   1:  PR[91,2] = PR[90,2] + -5.952;
   1:  PR[91,3] = PR[90,3] + 71.100;
   1:L PR[91] R[100]mm/sec CNT100;
   1:  PR[91,1] = PR[90,1] + 75.021;
   1:  PR[91,2] = PR[90,2] + -5.106;
   1:  PR[91,3] = PR[90,3] + 71.120;
   1:L PR[91] R[100]mm/sec CNT100;
   1:  PR[91,1] = PR[90,1] + 75.710;
   1:  PR[91,2] = PR[90,2] + -0.815;
   1:  PR[91,3] = PR[90,3] + 71.123;
   1:L PR[91] R[100]mm/sec CNT100;
   1:  PR[91,1] = PR[90,1] + 75.480;
   1:  PR[91,2] = PR[90,2] + 0.111;
   1:  PR[91,3] = PR[90,3] + 71.139;
   1:L PR[91] R[100]mm/sec CNT100;
   1:  PR[91,1] = PR[90,1] + 74.909;
   1:  PR[91,2] = PR[90,2] + 4.493;
   1:  PR[91,3] = PR[90,3] + 71.143;
   1:L PR[91] R[100]mm/sec CNT100;
   1:  PR[91,1] = PR[90,1] + 72.862;
   1:  PR[91,2] = PR[90,2] + 9.573;
   1:  PR[91,3] = PR[90,3] + 71.159;
   1:L PR[91] R[100]mm/sec CNT100;
   1:  PR[91,1] = PR[90,1] + 71.941;
   1:  PR[91,2] = PR[90,2] + 10.859;
   1:  PR[91,3] = PR[90,3] + 71.179;
   1:L PR[91] R[100]mm/sec CNT100;
   1:  PR[91,1] = PR[90,1] + 69.608;
   1:  PR[91,2] = PR[90,2] + 13.845;
   1:  PR[91,3] = PR[90,3] + 71.185;
   1:L PR[91] R[100]mm/sec CNT100;
   1:  PR[91,1] = PR[90,1] + 69.298;
   1:  PR[91,2] = PR[90,2] + 14.226;
   1:  PR[91,3] = PR[90,3] + 71.199;
   1:L PR[91] R[100]mm/sec CNT100;
   1:  PR[91,1] = PR[90,1] + 68.582;
   1:  PR[91,2] = PR[90,2] + 14.856;
   1:  PR[91,3] = PR[90,3] + 71.201;
   1:L PR[91] R[100]mm/sec CNT100;
   1:  PR[91,1] = PR[90,1] + 64.894;
   1:  PR[91,2] = PR[90,2] + 17.899;
   1:  PR[91,3] = PR[90,3] + 71.204;
   1:L PR[91] R[100]mm/sec CNT100;
   1:  PR[91,1] = PR[90,1] + 62.420;
   1:  PR[91,2] = PR[90,2] + 19.477;
   1:  PR[91,3] = PR[90,3] + 71.222;
   1:L PR[91] R[100]mm/sec CNT100;
   1:  PR[91,1] = PR[90,1] + 60.608;
   1:  PR[91,2] = PR[90,2] + 20.459;
   1:  PR[91,3] = PR[90,3] + 71.233;
   1:L PR[91] R[100]mm/sec CNT100;
   1:  PR[91,1] = PR[90,1] + 56.591;
   1:  PR[91,2] = PR[90,2] + 22.307;
   1:  PR[91,3] = PR[90,3] + 71.240;
   1:L PR[91] R[100]mm/sec CNT100;
   1:  PR[91,1] = PR[90,1] + 54.711;
   1:  PR[91,2] = PR[90,2] + 22.922;
   1:  PR[91,3] = PR[90,3] + 71.256;
   1:L PR[91] R[100]mm/sec CNT100;
   1:  PR[91,1] = PR[90,1] + 52.146;
   1:  PR[91,2] = PR[90,2] + 23.718;
   1:  PR[91,3] = PR[90,3] + 71.264;
   1:L PR[91] R[100]mm/sec CNT100;
   1:  PR[91,1] = PR[90,1] + 51.088;
   1:  PR[91,2] = PR[90,2] + 23.935;
   1:  PR[91,3] = PR[90,3] + 71.274;
   1:L PR[91] R[100]mm/sec CNT100;
   1:  PR[91,1] = PR[90,1] + 47.420;
   1:  PR[91,2] = PR[90,2] + 24.845;
   1:  PR[91,3] = PR[90,3] + 71.278;
   1:L PR[91] R[100]mm/sec CNT100;
   1:  PR[91,1] = PR[90,1] + 42.741;
   1:  PR[91,2] = PR[90,2] + 25.473;
   1:  PR[91,3] = PR[90,3] + 71.291;
   1:L PR[91] R[100]mm/sec CNT100;
   1:  PR[91,1] = PR[90,1] + 41.965;
   1:  PR[91,2] = PR[90,2] + 25.566;
   1:  PR[91,3] = PR[90,3] + 71.309;
   1:L PR[91] R[100]mm/sec CNT100;
   1:  PR[91,1] = PR[90,1] + 41.084;
   1:  PR[91,2] = PR[90,2] + 25.570;
   1:  PR[91,3] = PR[90,3] + 71.312;
   1:L PR[91] R[100]mm/sec CNT100;
   1:  PR[91,1] = PR[90,1] + 37.170;
   1:  PR[91,2] = PR[90,2] + 25.636;
   1:  PR[91,3] = PR[90,3] + 71.315;
   1:L PR[91] R[100]mm/sec CNT100;
   1:  PR[91,1] = PR[90,1] + 34.823;
   1:  PR[91,2] = PR[90,2] + 25.445;
   1:  PR[91,3] = PR[90,3] + 71.329;
   1:L PR[91] R[100]mm/sec CNT100;
   1:  PR[91,1] = PR[90,1] + 32.347;
   1:  PR[91,2] = PR[90,2] + 25.103;
   1:  PR[91,3] = PR[90,3] + 71.338;
   1:L PR[91] R[100]mm/sec CNT100;
   1:  PR[91,1] = PR[90,1] + 27.084;
   1:  PR[91,2] = PR[90,2] + 23.838;
   1:  PR[91,3] = PR[90,3] + 71.347;
   1:L PR[91] R[100]mm/sec CNT100;
   1:  PR[91,1] = PR[90,1] + 22.919;
   1:  PR[91,2] = PR[90,2] + 24.474;
   1:  PR[91,3] = PR[90,3] + 71.367;
   1:L PR[91] R[100]mm/sec CNT100;
   1:  PR[91,1] = PR[90,1] + 20.600;
   1:  PR[91,2] = PR[90,2] + 24.549;
   1:  PR[91,3] = PR[90,3] + 71.382;
   1:L PR[91] R[100]mm/sec CNT100;
   1:  PR[91,1] = PR[90,1] + 17.020;
   1:  PR[91,2] = PR[90,2] + 24.403;
   1:  PR[91,3] = PR[90,3] + 71.391;
   1:L PR[91] R[100]mm/sec CNT100;
   1:  PR[91,1] = PR[90,1] + 14.351;
   1:  PR[91,2] = PR[90,2] + 23.828;
   1:  PR[91,3] = PR[90,3] + 71.404;
   1:L PR[91] R[100]mm/sec CNT100;
   1:  PR[91,1] = PR[90,1] + 11.204;
   1:  PR[91,2] = PR[90,2] + 22.970;
   1:  PR[91,3] = PR[90,3] + 71.414;
   1:L PR[91] R[100]mm/sec CNT100;
   1:  PR[91,1] = PR[90,1] + 7.848;
   1:  PR[91,2] = PR[90,2] + 21.430;
   1:  PR[91,3] = PR[90,3] + 71.426;
   1:L PR[91] R[100]mm/sec CNT100;
   1:  PR[91,1] = PR[90,1] + 3.303;
   1:  PR[91,2] = PR[90,2] + 22.600;
   1:  PR[91,3] = PR[90,3] + 71.440;
   1:L PR[91] R[100]mm/sec CNT100;
   1:  PR[91,1] = PR[90,1] + 1.714;
   1:  PR[91,2] = PR[90,2] + 23.052;
   1:  PR[91,3] = PR[90,3] + 71.457;
   1:L PR[91] R[100]mm/sec CNT100;
   1:  PR[91,1] = PR[90,1] + -4.595;
   1:  PR[91,2] = PR[90,2] + 23.619;
   1:  PR[91,3] = PR[90,3] + 71.463;
   1:L PR[91] R[100]mm/sec CNT100;
   1:  PR[91,1] = PR[90,1] + -7.696;
   1:  PR[91,2] = PR[90,2] + 23.369;
   1:  PR[91,3] = PR[90,3] + 71.486;
   1:L PR[91] R[100]mm/sec CNT100;
   1:  PR[91,1] = PR[90,1] + -10.709;
   1:  PR[91,2] = PR[90,2] + 23.080;
   1:  PR[91,3] = PR[90,3] + 71.498;
   1:L PR[91] R[100]mm/sec CNT100;
   1:  PR[91,1] = PR[90,1] + -13.600;
   1:  PR[91,2] = PR[90,2] + 22.402;
   1:  PR[91,3] = PR[90,3] + 71.509;
   1:L PR[91] R[100]mm/sec CNT100;
   1:  PR[91,1] = PR[90,1] + -15.931;
   1:  PR[91,2] = PR[90,2] + 21.755;
   1:  PR[91,3] = PR[90,3] + 71.520;
   1:L PR[91] R[100]mm/sec CNT100;
   1:  PR[91,1] = PR[90,1] + -17.870;
   1:  PR[91,2] = PR[90,2] + 22.083;
   1:  PR[91,3] = PR[90,3] + 71.529;
   1:L PR[91] R[100]mm/sec CNT100;
   1:  PR[91,1] = PR[90,1] + -19.775;
   1:  PR[91,2] = PR[90,2] + 22.343;
   1:  PR[91,3] = PR[90,3] + 71.536;
   1:L PR[91] R[100]mm/sec CNT100;
   1:  PR[91,1] = PR[90,1] + -26.709;
   1:  PR[91,2] = PR[90,2] + 23.102;
   1:  PR[91,3] = PR[90,3] + 71.543;
   1:L PR[91] R[100]mm/sec CNT100;
   1:  PR[91,1] = PR[90,1] + -27.634;
   1:  PR[91,2] = PR[90,2] + 23.219;
   1:  PR[91,3] = PR[90,3] + 71.569;
   1:L PR[91] R[100]mm/sec CNT100;
   1:  PR[91,1] = PR[90,1] + -35.837;
   1:  PR[91,2] = PR[90,2] + 23.471;
   1:  PR[91,3] = PR[90,3] + 71.572;
   1:L PR[91] R[100]mm/sec CNT100;
   1:  PR[91,1] = PR[90,1] + -37.663;
   1:  PR[91,2] = PR[90,2] + 23.575;
   1:  PR[91,3] = PR[90,3] + 71.602;
   1:L PR[91] R[100]mm/sec CNT100;
   1:  PR[91,1] = PR[90,1] + -41.865;
   1:  PR[91,2] = PR[90,2] + 23.392;
   1:  PR[91,3] = PR[90,3] + 71.609;
   1:L PR[91] R[100]mm/sec CNT100;
   1:  PR[91,1] = PR[90,1] + -44.716;
   1:  PR[91,2] = PR[90,2] + 23.204;
   1:  PR[91,3] = PR[90,3] + 71.624;
   1:L PR[91] R[100]mm/sec CNT100;
   1:  PR[91,1] = PR[90,1] + -50.383;
   1:  PR[91,2] = PR[90,2] + 22.257;
   1:  PR[91,3] = PR[90,3] + 71.635;
   1:L PR[91] R[100]mm/sec CNT100;
   1:  PR[91,1] = PR[90,1] + -53.393;
   1:  PR[91,2] = PR[90,2] + 21.640;
   1:  PR[91,3] = PR[90,3] + 71.656;
   1:L PR[91] R[100]mm/sec CNT100;
   1:  PR[91,1] = PR[90,1] + -55.296;
   1:  PR[91,2] = PR[90,2] + 21.017;
   1:  PR[91,3] = PR[90,3] + 71.667;
   1:L PR[91] R[100]mm/sec CNT100;
   1:  PR[91,1] = PR[90,1] + -58.574;
   1:  PR[91,2] = PR[90,2] + 19.824;
   1:  PR[91,3] = PR[90,3] + 71.675;
   1:L PR[91] R[100]mm/sec CNT100;
   1:  PR[91,1] = PR[90,1] + -60.495;
   1:  PR[91,2] = PR[90,2] + 19.070;
   1:  PR[91,3] = PR[90,3] + 71.687;
   1:L PR[91] R[100]mm/sec CNT100;
   1:  PR[91] = PR[90];
   1:  PR[91,1] = PR[90,1] + -64.658;
   1:  PR[91,2] = PR[90,2] + 16.036;
   1:  PR[91,3] = PR[90,3] + 72.995;
   1:L PR[91] R[100]mm/sec CNT100;
   1:  PR[91,1] = PR[90,1] + -66.807;
   1:  PR[91,2] = PR[90,2] + 14.084;
   1:  PR[91,3] = PR[90,3] + 71.717;
   1:L PR[91] R[100]mm/sec CNT100;
   1:  PR[91,1] = PR[90,1] + -68.784;
   1:  PR[91,2] = PR[90,2] + 12.271;
   1:  PR[91,3] = PR[90,3] + 71.728;
   1:L PR[91] R[100]mm/sec CNT100;
   1:  PR[91,1] = PR[90,1] + -71.738;
   1:  PR[91,2] = PR[90,2] + 8.120;
   1:  PR[91,3] = PR[90,3] + 71.738;
   1:L PR[91] R[100]mm/sec CNT100;
   1:  PR[91,1] = PR[90,1] + -73.499;
   1:  PR[91,2] = PR[90,2] + 3.745;
   1:  PR[91,3] = PR[90,3] + 71.757;
   1:L PR[91] R[100]mm/sec CNT100;
   1:  PR[91,1] = PR[90,1] + -74.080;
   1:  PR[91,2] = PR[90,2] + -0.689;
   1:  PR[91,3] = PR[90,3] + 71.774;
   1:L PR[91] R[100]mm/sec CNT100;
   1:  PR[91,1] = PR[90,1] + -73.575;
   1:  PR[91,2] = PR[90,2] + -3.117;
   1:  PR[91,3] = PR[90,3] + 71.791;
   1:L PR[91] R[100]mm/sec CNT100;
   1:  PR[91,1] = PR[90,1] + -73.284;
   1:  PR[91,2] = PR[90,2] + -5.386;
   1:  PR[91,3] = PR[90,3] + 71.800;
   1:L PR[91] R[100]mm/sec CNT100;
   1:  PR[91,1] = PR[90,1] + -72.278;
   1:  PR[91,2] = PR[90,2] + -7.892;
   1:  PR[91,3] = PR[90,3] + 71.808;
   1:L PR[91] R[100]mm/sec CNT100;
   1:  PR[91,1] = PR[90,1] + -71.464;
   1:  PR[91,2] = PR[90,2] + -9.892;
   1:  PR[91,3] = PR[90,3] + 71.818;
   1:L PR[91] R[100]mm/sec CNT100;
   1:  PR[91,1] = PR[90,1] + -68.451;
   1:  PR[91,2] = PR[90,2] + -14.108;
   1:  PR[91,3] = PR[90,3] + 71.826;
   1:L PR[91] R[100]mm/sec CNT100;
   1:  PR[91,1] = PR[90,1] + -64.359;
   1:  PR[91,2] = PR[90,2] + -17.817;
   1:  PR[91,3] = PR[90,3] + 71.846;
   1:L PR[91] R[100]mm/sec CNT100;
   1:  PR[91,1] = PR[90,1] + -59.208;
   1:  PR[91,2] = PR[90,2] + -20.687;
   1:  PR[91,3] = PR[90,3] + 71.866;
   1:L PR[91] R[100]mm/sec CNT100;
   1:  PR[91,1] = PR[90,1] + -56.302;
   1:  PR[91,2] = PR[90,2] + -21.871;
   1:  PR[91,3] = PR[90,3] + 71.888;
   1:L PR[91] R[100]mm/sec CNT100;
   1:  PR[91,1] = PR[90,1] + -53.674;
   1:  PR[91,2] = PR[90,2] + -22.806;
   1:  PR[91,3] = PR[90,3] + 71.900;
   1:L PR[91] R[100]mm/sec CNT100;
   1:  PR[91,1] = PR[90,1] + -49.742;
   1:  PR[91,2] = PR[90,2] + -23.757;
   1:  PR[91,3] = PR[90,3] + 71.910;
   1:L PR[91] R[100]mm/sec CNT100;
   1:  PR[91,1] = PR[90,1] + -47.986;
   1:  PR[91,2] = PR[90,2] + -24.162;
   1:  PR[91,3] = PR[90,3] + 71.925;
   1:L PR[91] R[100]mm/sec CNT100;
   1:  PR[91,1] = PR[90,1] + -46.736;
   1:  PR[91,2] = PR[90,2] + -24.408;
   1:  PR[91,3] = PR[90,3] + 71.932;
   1:L PR[91] R[100]mm/sec CNT100;
   1:  PR[91,1] = PR[90,1] + -42.499;
   1:  PR[91,2] = PR[90,2] + -24.853;
   1:  PR[91,3] = PR[90,3] + 71.937;
   1:L PR[91] R[100]mm/sec CNT100;
   1:  PR[91,1] = PR[90,1] + -37.572;
   1:  PR[91,2] = PR[90,2] + -25.182;
   1:  PR[91,3] = PR[90,3] + 71.952;
   1:L PR[91] R[100]mm/sec CNT100;
   1:  PR[91,1] = PR[90,1] + -36.488;
   1:  PR[91,2] = PR[90,2] + -25.268;
   1:  PR[91,3] = PR[90,3] + 71.971;
   1:L PR[91] R[100]mm/sec CNT100;
   1:  PR[91,1] = PR[90,1] + -35.528;
   1:  PR[91,2] = PR[90,2] + -25.297;
   1:  PR[91,3] = PR[90,3] + 71.975;
   1:L PR[91] R[100]mm/sec CNT100;
   1:  PR[91,1] = PR[90,1] + -30.632;
   1:  PR[91,2] = PR[90,2] + -25.146;
   1:  PR[91,3] = PR[90,3] + 71.978;
   1:L PR[91] R[100]mm/sec CNT100;
   1:  PR[91,1] = PR[90,1] + -24.961;
   1:  PR[91,2] = PR[90,2] + -24.930;
   1:  PR[91,3] = PR[90,3] + 71.996;
   1:L PR[91] R[100]mm/sec CNT100;
   1:  PR[91,1] = PR[90,1] + -17.966;
   1:  PR[91,2] = PR[90,2] + -24.135;
   1:  PR[91,3] = PR[90,3] + 72.017;
   1:L PR[91] R[100]mm/sec CNT100;
   1:  PR[91,1] = PR[90,1] + -17.484;
   1:  PR[91,2] = PR[90,2] + -24.120;
   1:  PR[91,3] = PR[90,3] + 72.044;
   1:L PR[91] R[100]mm/sec CNT100;
   1:  PR[91,1] = PR[90,1] + -14.422;
   1:  PR[91,2] = PR[90,2] + -23.701;
   1:  PR[91,3] = PR[90,3] + 72.045;
   1:L PR[91] R[100]mm/sec CNT100;
   1:  PR[91,1] = PR[90,1] + -10.015;
   1:  PR[91,2] = PR[90,2] + -24.736;
   1:  PR[91,3] = PR[90,3] + 72.057;
   1:L PR[91] R[100]mm/sec CNT100;
   1:  PR[91,1] = PR[90,1] + -5.899;
   1:  PR[91,2] = PR[90,2] + -25.133;
   1:  PR[91,3] = PR[90,3] + 72.074;
   1:L PR[91] R[100]mm/sec CNT100;
   1:  PR[91,1] = PR[90,1] + -3.854;
   1:  PR[91,2] = PR[90,2] + -25.298;
   1:  PR[91,3] = PR[90,3] + 72.089;
   1:L PR[91] R[100]mm/sec CNT100;
   1:  PR[91,1] = PR[90,1] + 2.663;
   1:  PR[91,2] = PR[90,2] + -24.737;
   1:  PR[91,3] = PR[90,3] + 72.097;
   1:L PR[91] R[100]mm/sec CNT100;
   1:  PR[91,1] = PR[90,1] + 8.196;
   1:  PR[91,2] = PR[90,2] + -23.321;
   1:  PR[91,3] = PR[90,3] + 72.121;
   1:L PR[91] R[100]mm/sec CNT100;
   1:  PR[91,1] = PR[90,1] + 11.071;
   1:  PR[91,2] = PR[90,2] + -24.641;
   1:  PR[91,3] = PR[90,3] + 72.142;
   1:L PR[91] R[100]mm/sec CNT100;
   1:  PR[91,1] = PR[90,1] + 13.655;
   1:  PR[91,2] = PR[90,2] + -25.345;
   1:  PR[91,3] = PR[90,3] + 72.154;
   1:L PR[91] R[100]mm/sec CNT100;
   1:  PR[91,1] = PR[90,1] + 16.983;
   1:  PR[91,2] = PR[90,2] + -26.063;
   1:  PR[91,3] = PR[90,3] + 72.164;
   1:L PR[91] R[100]mm/sec CNT100;
   1:  PR[91,1] = PR[90,1] + 19.995;
   1:  PR[91,2] = PR[90,2] + -26.185;
   1:  PR[91,3] = PR[90,3] + 72.176;
   1:L PR[91] R[100]mm/sec CNT100;
   1:  PR[91,1] = PR[90,1] + 22.970;
   1:  PR[91,2] = PR[90,2] + -26.089;
   1:  PR[91,3] = PR[90,3] + 72.188;
   1:L PR[91] R[100]mm/sec CNT100;
   1:  PR[91,1] = PR[90,1] + 26.634;
   1:  PR[91,2] = PR[90,2] + -25.533;
   1:  PR[91,3] = PR[90,3] + 72.199;
   1:L PR[91] R[100]mm/sec CNT100;
   1:  PR[91,1] = PR[90,1] + 29.088;
   1:  PR[91,2] = PR[90,2] + -26.173;
   1:  PR[91,3] = PR[90,3] + 72.212;
   1:L PR[91] R[100]mm/sec CNT100;
   1:  PR[91,1] = PR[90,1] + 31.868;
   1:  PR[91,2] = PR[90,2] + -26.840;
   1:  PR[91,3] = PR[90,3] + 72.222;
   1:L PR[91] R[100]mm/sec CNT100;
   1:  PR[91,1] = PR[90,1] + 33.215;
   1:  PR[91,2] = PR[90,2] + -27.027;
   1:  PR[91,3] = PR[90,3] + 72.232;
   1:L PR[91] R[100]mm/sec CNT100;
   1:  PR[91,1] = PR[90,1] + 36.811;
   1:  PR[91,2] = PR[90,2] + -27.319;
   1:  PR[91,3] = PR[90,3] + 72.237;
   1:L PR[91] R[100]mm/sec CNT100;
   1:  PR[91,1] = PR[90,1] + 40.668;
   1:  PR[91,2] = PR[90,2] + -27.254;
   1:  PR[91,3] = PR[90,3] + 72.251;
   1:L PR[91] R[100]mm/sec CNT100;
   1:  PR[91,1] = PR[90,1] + 41.328;
   1:  PR[91,2] = PR[90,2] + -27.203;
   1:  PR[91,3] = PR[90,3] + 72.265;
   1:L PR[91] R[100]mm/sec CNT100;
   1:  PR[91,1] = PR[90,1] + 42.439;
   1:  PR[91,2] = PR[90,2] + -27.011;
   1:  PR[91,3] = PR[90,3] + 72.268;
   1:L PR[91] R[100]mm/sec CNT100;
   1:  PR[91,1] = PR[90,1] + 46.630;
   1:  PR[91,2] = PR[90,2] + -26.449;
   1:  PR[91,3] = PR[90,3] + 72.272;
   1:L PR[91] R[100]mm/sec CNT100;
   1:  PR[91,1] = PR[90,1] + 50.455;
   1:  PR[91,2] = PR[90,2] + -25.500;
   1:  PR[91,3] = PR[90,3] + 72.288;
   1:L PR[91] R[100]mm/sec CNT100;
   1:  PR[91,1] = PR[90,1] + 51.336;
   1:  PR[91,2] = PR[90,2] + -25.262;
   1:  PR[91,3] = PR[90,3] + 72.302;
   1:L PR[91] R[100]mm/sec CNT100;
   1:  PR[91,1] = PR[90,1] + 52.051;
   1:  PR[91,2] = PR[90,2] + -24.984;
   1:  PR[91,3] = PR[90,3] + 72.306;
   1:L PR[91] R[100]mm/sec CNT100;
   1:  PR[91,1] = PR[90,1] + 55.819;
   1:  PR[91,2] = PR[90,2] + -23.752;
   1:  PR[91,3] = PR[90,3] + 72.308;
   1:L PR[91] R[100]mm/sec CNT100;
   1:  PR[91,1] = PR[90,1] + 60.017;
   1:  PR[91,2] = PR[90,2] + -21.841;
   1:  PR[91,3] = PR[90,3] + 72.323;
   1:L PR[91] R[100]mm/sec CNT100;
   1:  PR[91,1] = PR[90,1] + 60.781;
   1:  PR[91,2] = PR[90,2] + -21.428;
   1:  PR[91,3] = PR[90,3] + 72.340;
   1:L PR[91] R[100]mm/sec CNT100;
   1:  PR[91,1] = PR[90,1] + 64.071;
   1:  PR[91,2] = PR[90,2] + -19.328;
   1:  PR[91,3] = PR[90,3] + 72.343;
   1:L PR[91] R[100]mm/sec CNT100;
   1:  PR[91,1] = PR[90,1] + 66.786;
   1:  PR[91,2] = PR[90,2] + -17.090;
   1:  PR[91,3] = PR[90,3] + 72.358;
   1:L PR[91] R[100]mm/sec CNT100;
   1:  PR[91,1] = PR[90,1] + 68.269;
   1:  PR[91,2] = PR[90,2] + -15.785;
   1:  PR[91,3] = PR[90,3] + 72.371;
   1:L PR[91] R[100]mm/sec CNT100;
   1:  PR[91,1] = PR[90,1] + 71.977;
   1:  PR[91,2] = PR[90,2] + -11.080;
   1:  PR[91,3] = PR[90,3] + 72.378;
   1:L PR[91] R[100]mm/sec CNT100;
   1:  PR[91,1] = PR[90,1] + 72.022;
   1:  PR[91,2] = PR[90,2] + -10.999;
   1:  PR[91,3] = PR[90,3] + 72.401;
   1:L PR[91] R[100]mm/sec CNT100;
   1:  PR[91,1] = PR[90,1] + 73.204;
   1:  PR[91,2] = PR[90,2] + -8.301;
   1:L PR[91] R[100]mm/sec CNT100;
   1:  PR[91,1] = PR[90,1] + 74.139;
   1:  PR[91,2] = PR[90,2] + -5.981;
   1:  PR[91,3] = PR[90,3] + 72.412;
   1:L PR[91] R[100]mm/sec CNT100;
   1:  PR[91,1] = PR[90,1] + 74.388;
   1:  PR[91,2] = PR[90,2] + -4.382;
   1:  PR[91,3] = PR[90,3] + 72.421;
   1:L PR[91] R[100]mm/sec CNT100;
   1:  PR[91,1] = PR[90,1] + 74.867;
   1:  PR[91,2] = PR[90,2] + -0.844;
   1:  PR[91,3] = PR[90,3] + 72.427;
   1:L PR[91] R[100]mm/sec CNT100;
   1:  PR[91,1] = PR[90,1] + 74.796;
   1:  PR[91,2] = PR[90,2] + -0.562;
   1:  PR[91,3] = PR[90,3] + 72.440;
   1:L PR[91] R[100]mm/sec CNT100;
   1:  PR[91,1] = PR[90,1] + 74.131;
   1:  PR[91,2] = PR[90,2] + 4.543;
   1:  PR[91,3] = PR[90,3] + 72.441;
   1:L PR[91] R[100]mm/sec CNT100;
   1:  PR[91,1] = PR[90,1] + 73.204;
   1:  PR[91,2] = PR[90,2] + 6.843;
   1:  PR[91,3] = PR[90,3] + 72.461;
   1:L PR[91] R[100]mm/sec CNT100;
   1:  PR[91,1] = PR[90,1] + 72.026;
   1:  PR[91,2] = PR[90,2] + 9.535;
   1:  PR[91,3] = PR[90,3] + 72.470;
   1:L PR[91] R[100]mm/sec CNT100;
   1:  PR[91,1] = PR[90,1] + 71.979;
   1:  PR[91,2] = PR[90,2] + 9.618;
   1:  PR[91,3] = PR[90,3] + 72.481;
   1:L PR[91] R[100]mm/sec CNT100;
   1:  PR[91,1] = PR[90,1] + 68.980;
   1:  PR[91,2] = PR[90,2] + 13.457;
   1:L PR[91] R[100]mm/sec CNT100;
   1:  PR[91,1] = PR[90,1] + 68.287;
   1:  PR[91,2] = PR[90,2] + 14.310;
   1:  PR[91,3] = PR[90,3] + 72.499;
   1:L PR[91] R[100]mm/sec CNT100;
   1:  PR[91,1] = PR[90,1] + 66.792;
   1:  PR[91,2] = PR[90,2] + 15.625;
   1:  PR[91,3] = PR[90,3] + 72.503;
   1:L PR[91] R[100]mm/sec CNT100;
   1:  PR[91,1] = PR[90,1] + 64.076;
   1:  PR[91,2] = PR[90,2] + 17.866;
   1:  PR[91,3] = PR[90,3] + 72.511;
   1:L PR[91] R[100]mm/sec CNT100;
   1:  PR[91,1] = PR[90,1] + 60.784;
   1:  PR[91,2] = PR[90,2] + 19.967;
   1:  PR[91,3] = PR[90,3] + 72.524;
   1:L PR[91] R[100]mm/sec CNT100;
   1:  PR[91,1] = PR[90,1] + 60.019;
   1:  PR[91,2] = PR[90,2] + 20.382;
   1:  PR[91,3] = PR[90,3] + 72.538;
   1:L PR[91] R[100]mm/sec CNT100;
   1:  PR[91,1] = PR[90,1] + 55.819;
   1:  PR[91,2] = PR[90,2] + 22.294;
   1:  PR[91,3] = PR[90,3] + 72.541;
   1:L PR[91] R[100]mm/sec CNT100;
   1:  PR[91,1] = PR[90,1] + 52.051;
   1:  PR[91,2] = PR[90,2] + 23.525;
   1:  PR[91,3] = PR[90,3] + 72.558;
   1:L PR[91] R[100]mm/sec CNT100;
   1:  PR[91,1] = PR[90,1] + 51.336;
   1:  PR[91,2] = PR[90,2] + 23.803;
   1:  PR[91,3] = PR[90,3] + 72.573;
   1:L PR[91] R[100]mm/sec CNT100;
   1:  PR[91,1] = PR[90,1] + 50.455;
   1:  PR[91,2] = PR[90,2] + 24.041;
   1:  PR[91,3] = PR[90,3] + 72.576;
   1:L PR[91] R[100]mm/sec CNT100;
   1:  PR[91,1] = PR[90,1] + 46.630;
   1:  PR[91,2] = PR[90,2] + 24.990;
   1:  PR[91,3] = PR[90,3] + 72.579;
   1:L PR[91] R[100]mm/sec CNT100;
   1:  PR[91,1] = PR[90,1] + 42.439;
   1:  PR[91,2] = PR[90,2] + 25.553;
   1:  PR[91,3] = PR[90,3] + 72.594;
   1:L PR[91] R[100]mm/sec CNT100;
   1:  PR[91,1] = PR[90,1] + 41.328;
   1:  PR[91,2] = PR[90,2] + 25.744;
   1:  PR[91,3] = PR[90,3] + 72.610;
   1:L PR[91] R[100]mm/sec CNT100;
   1:  PR[91,1] = PR[90,1] + 40.668;
   1:  PR[91,2] = PR[90,2] + 25.795;
   1:  PR[91,3] = PR[90,3] + 72.614;
   1:L PR[91] R[100]mm/sec CNT100;
   1:  PR[91,1] = PR[90,1] + 36.811;
   1:  PR[91,2] = PR[90,2] + 25.860;
   1:  PR[91,3] = PR[90,3] + 72.616;
   1:L PR[91] R[100]mm/sec CNT100;
   1:  PR[91,1] = PR[90,1] + 33.215;
   1:  PR[91,2] = PR[90,2] + 25.568;
   1:  PR[91,3] = PR[90,3] + 72.631;
   1:L PR[91] R[100]mm/sec CNT100;
   1:  PR[91,1] = PR[90,1] + 31.868;
   1:  PR[91,2] = PR[90,2] + 25.382;
   1:  PR[91,3] = PR[90,3] + 72.644;
   1:L PR[91] R[100]mm/sec CNT100;
   1:  PR[91,1] = PR[90,1] + 29.088;
   1:  PR[91,2] = PR[90,2] + 24.714;
   1:  PR[91,3] = PR[90,3] + 72.649;
   1:L PR[91] R[100]mm/sec CNT100;
   1:  PR[91,1] = PR[90,1] + 26.634;
   1:  PR[91,2] = PR[90,2] + 24.074;
   1:  PR[91,3] = PR[90,3] + 72.660;
   1:L PR[91] R[100]mm/sec CNT100;
   1:  PR[91,1] = PR[90,1] + 22.970;
   1:  PR[91,2] = PR[90,2] + 24.630;
   1:  PR[91,3] = PR[90,3] + 72.669;
   1:L PR[91] R[100]mm/sec CNT100;
   1:  PR[91,1] = PR[90,1] + 19.995;
   1:  PR[91,2] = PR[90,2] + 24.726;
   1:  PR[91,3] = PR[90,3] + 72.683;
   1:L PR[91] R[100]mm/sec CNT100;
   1:  PR[91,1] = PR[90,1] + 16.982;
   1:  PR[91,2] = PR[90,2] + 24.604;
   1:  PR[91,3] = PR[90,3] + 72.694;
   1:L PR[91] R[100]mm/sec CNT100;
   1:  PR[91,1] = PR[90,1] + 13.654;
   1:  PR[91,2] = PR[90,2] + 23.886;
   1:  PR[91,3] = PR[90,3] + 72.705;
   1:L PR[91] R[100]mm/sec CNT100;
   1:  PR[91,1] = PR[90,1] + 11.070;
   1:  PR[91,2] = PR[90,2] + 23.182;
   1:  PR[91,3] = PR[90,3] + 72.718;
   1:L PR[91] R[100]mm/sec CNT100;
   1:  PR[91,1] = PR[90,1] + 8.194;
   1:  PR[91,2] = PR[90,2] + 21.862;
   1:  PR[91,3] = PR[90,3] + 72.728;
   1:L PR[91] R[100]mm/sec CNT100;
   1:  PR[91,1] = PR[90,1] + 2.710;
   1:  PR[91,2] = PR[90,2] + 23.270;
   1:  PR[91,3] = PR[90,3] + 72.739;
   1:L PR[91] R[100]mm/sec CNT100;
   1:  PR[91,1] = PR[90,1] + -3.833;
   1:  PR[91,2] = PR[90,2] + 23.839;
   1:  PR[91,3] = PR[90,3] + 72.760;
   1:L PR[91] R[100]mm/sec CNT100;
   1:  PR[91,1] = PR[90,1] + -5.873;
   1:  PR[91,2] = PR[90,2] + 23.675;
   1:  PR[91,3] = PR[90,3] + 72.785;
   1:L PR[91] R[100]mm/sec CNT100;
   1:  PR[91,1] = PR[90,1] + -10.012;
   1:  PR[91,2] = PR[90,2] + 23.278;
   1:  PR[91,3] = PR[90,3] + 72.792;
   1:L PR[91] R[100]mm/sec CNT100;
   1:  PR[91,1] = PR[90,1] + -14.423;
   1:  PR[91,2] = PR[90,2] + 22.242;
   1:  PR[91,3] = PR[90,3] + 72.808;
   1:L PR[91] R[100]mm/sec CNT100;
   1:  PR[91,1] = PR[90,1] + -17.559;
   1:  PR[91,2] = PR[90,2] + 22.671;
   1:  PR[91,3] = PR[90,3] + 72.825;
   1:L PR[91] R[100]mm/sec CNT100;
   1:  PR[91,1] = PR[90,1] + -24.454;
   1:  PR[91,2] = PR[90,2] + 23.425;
   1:  PR[91,3] = PR[90,3] + 72.836;
   1:L PR[91] R[100]mm/sec CNT100;
   1:  PR[91,1] = PR[90,1] + -24.988;
   1:  PR[91,2] = PR[90,2] + 23.474;
   1:  PR[91,3] = PR[90,3] + 72.862;
   1:L PR[91] R[100]mm/sec CNT100;
   1:  PR[91,1] = PR[90,1] + -27.189;
   1:  PR[91,2] = PR[90,2] + 23.557;
   1:  PR[91,3] = PR[90,3] + 72.864;
   1:L PR[91] R[100]mm/sec CNT100;
   1:  PR[91,1] = PR[90,1] + -36.501;
   1:  PR[91,2] = PR[90,2] + 23.825;
   1:  PR[91,3] = PR[90,3] + 72.872;
   1:L PR[91] R[100]mm/sec CNT100;
   1:  PR[91,1] = PR[90,1] + -43.578;
   1:  PR[91,2] = PR[90,2] + 23.358;
   1:  PR[91,3] = PR[90,3] + 72.907;
   1:L PR[91] R[100]mm/sec CNT100;
   1:  PR[91,1] = PR[90,1] + -49.857;
   1:  PR[91,2] = PR[90,2] + 22.298;
   1:  PR[91,3] = PR[90,3] + 72.933;
   1:L PR[91] R[100]mm/sec CNT100;
   1:  PR[91,1] = PR[90,1] + -51.705;
   1:  PR[91,2] = PR[90,2] + 21.919;
   1:  PR[91,3] = PR[90,3] + 72.957;
   1:L PR[91] R[100]mm/sec CNT100;
   1:  PR[91,1] = PR[90,1] + -54.751;
   1:  PR[91,2] = PR[90,2] + 20.923;
   1:  PR[91,3] = PR[90,3] + 72.964;
   1:L PR[91] R[100]mm/sec CNT100;
   1:  PR[91,1] = PR[90,1] + -59.398;
   1:  PR[91,2] = PR[90,2] + 19.232;
   1:  PR[91,3] = PR[90,3] + 72.976;
   1:L PR[91] R[100]mm/sec CNT100;
   1:  PR[91,1] = PR[90,1] + -59.600;
   1:  PR[91,2] = PR[90,2] + 19.121;
   1:  PR[91,3] = PR[90,3] + 72.994;
   1:L PR[91] R[100]mm/sec CNT100;
   1:  PR[91] = PR[90];
   1:  PR[91,1] = PR[90,1] + -60.911;
   1:  PR[91,2] = PR[90,2] + 17.831;
   1:  PR[91,3] = PR[90,3] + 74.295;
   1:L PR[91] R[100]mm/sec CNT100;
   1:  PR[91,1] = PR[90,1] + -63.605;
   1:  PR[91,2] = PR[90,2] + 16.188;
   1:  PR[91,3] = PR[90,3] + 73.004;
   1:L PR[91] R[100]mm/sec CNT100;
   1:  PR[91,1] = PR[90,1] + -67.777;
   1:  PR[91,2] = PR[90,2] + 12.385;
   1:  PR[91,3] = PR[90,3] + 73.016;
   1:L PR[91] R[100]mm/sec CNT100;
   1:  PR[91,1] = PR[90,1] + -70.758;
   1:  PR[91,2] = PR[90,2] + 8.199;
   1:  PR[91,3] = PR[90,3] + 73.037;
   1:L PR[91] R[100]mm/sec CNT100;
   1:  PR[91,1] = PR[90,1] + -72.537;
   1:  PR[91,2] = PR[90,2] + 3.785;
   1:  PR[91,3] = PR[90,3] + 73.056;
   1:L PR[91] R[100]mm/sec CNT100;
   1:  PR[91,1] = PR[90,1] + -73.033;
   1:  PR[91,2] = PR[90,2] + -0.004;
   1:  PR[91,3] = PR[90,3] + 73.074;
   1:L PR[91] R[100]mm/sec CNT100;
   1:  PR[91,1] = PR[90,1] + -73.156;
   1:  PR[91,2] = PR[90,2] + -0.698;
   1:  PR[91,3] = PR[90,3] + 73.089;
   1:L PR[91] R[100]mm/sec CNT100;
   1:  PR[91,1] = PR[90,1] + -72.777;
   1:  PR[91,2] = PR[90,2] + -2.521;
   1:  PR[91,3] = PR[90,3] + 73.091;
   1:L PR[91] R[100]mm/sec CNT100;
   1:  PR[91,1] = PR[90,1] + -72.405;
   1:  PR[91,2] = PR[90,2] + -5.414;
   1:  PR[91,3] = PR[90,3] + 73.098;
   1:L PR[91] R[100]mm/sec CNT100;
   1:  PR[91,1] = PR[90,1] + -71.119;
   1:  PR[91,2] = PR[90,2] + -8.619;
   1:  PR[91,3] = PR[90,3] + 73.109;
   1:L PR[91] R[100]mm/sec CNT100;
   1:  PR[91,1] = PR[90,1] + -70.578;
   1:  PR[91,2] = PR[90,2] + -9.947;
   1:  PR[91,3] = PR[90,3] + 73.122;
   1:L PR[91] R[100]mm/sec CNT100;
   1:  PR[91,1] = PR[90,1] + -67.553;
   1:  PR[91,2] = PR[90,2] + -14.191;
   1:  PR[91,3] = PR[90,3] + 73.127;
   1:L PR[91] R[100]mm/sec CNT100;
   1:  PR[91,1] = PR[90,1] + -65.728;
   1:  PR[91,2] = PR[90,2] + -15.844;
   1:  PR[91,3] = PR[90,3] + 73.147;
   1:L PR[91] R[100]mm/sec CNT100;
   1:  PR[91,1] = PR[90,1] + -63.351;
   1:  PR[91,2] = PR[90,2] + -17.826;
   1:  PR[91,3] = PR[90,3] + 73.156;
   1:L PR[91] R[100]mm/sec CNT100;
   1:  PR[91,1] = PR[90,1] + -62.402;
   1:  PR[91,2] = PR[90,2] + -18.408;
   1:  PR[91,3] = PR[90,3] + 73.168;
   1:L PR[91] R[100]mm/sec CNT100;
   1:  PR[91,1] = PR[90,1] + -58.268;
   1:  PR[91,2] = PR[90,2] + -20.710;
   1:  PR[91,3] = PR[90,3] + 73.172;
   1:L PR[91] R[100]mm/sec CNT100;
   1:  PR[91,1] = PR[90,1] + -54.059;
   1:  PR[91,2] = PR[90,2] + -22.425;
   1:  PR[91,3] = PR[90,3] + 73.190;
   1:L PR[91] R[100]mm/sec CNT100;
   1:  PR[91,1] = PR[90,1] + -52.795;
   1:  PR[91,2] = PR[90,2] + -22.875;
   1:  PR[91,3] = PR[90,3] + 73.207;
   1:L PR[91] R[100]mm/sec CNT100;
   1:  PR[91,1] = PR[90,1] + -50.854;
   1:  PR[91,2] = PR[90,2] + -23.345;
   1:  PR[91,3] = PR[90,3] + 73.212;
   1:L PR[91] R[100]mm/sec CNT100;
   1:  PR[91,1] = PR[90,1] + -47.243;
   1:  PR[91,2] = PR[90,2] + -24.177;
   1:  PR[91,3] = PR[90,3] + 73.219;
   1:L PR[91] R[100]mm/sec CNT100;
   1:  PR[91,1] = PR[90,1] + -44.582;
   1:  PR[91,2] = PR[90,2] + -24.700;
   1:  PR[91,3] = PR[90,3] + 73.233;
   1:L PR[91] R[100]mm/sec CNT100;
   1:  PR[91,1] = PR[90,1] + -41.757;
   1:  PR[91,2] = PR[90,2] + -24.997;
   1:  PR[91,3] = PR[90,3] + 73.243;
   1:L PR[91] R[100]mm/sec CNT100;
   1:  PR[91,1] = PR[90,1] + -38.433;
   1:  PR[91,2] = PR[90,2] + -25.218;
   1:  PR[91,3] = PR[90,3] + 73.254;
   1:L PR[91] R[100]mm/sec CNT100;
   1:  PR[91,1] = PR[90,1] + -35.329;
   1:  PR[91,2] = PR[90,2] + -25.466;
   1:  PR[91,3] = PR[90,3] + 73.266;
   1:L PR[91] R[100]mm/sec CNT100;
   1:  PR[91,1] = PR[90,1] + -32.441;
   1:  PR[91,2] = PR[90,2] + -25.552;
   1:  PR[91,3] = PR[90,3] + 73.278;
   1:L PR[91] R[100]mm/sec CNT100;
   1:  PR[91,1] = PR[90,1] + -29.752;
   1:  PR[91,2] = PR[90,2] + -25.470;
   1:  PR[91,3] = PR[90,3] + 73.289;
   1:L PR[91] R[100]mm/sec CNT100;
   1:  PR[91,1] = PR[90,1] + -22.134;
   1:  PR[91,2] = PR[90,2] + -25.177;
   1:  PR[91,3] = PR[90,3] + 73.299;
   1:L PR[91] R[100]mm/sec CNT100;
   1:  PR[91,1] = PR[90,1] + -15.897;
   1:  PR[91,2] = PR[90,2] + -24.469;
   1:  PR[91,3] = PR[90,3] + 73.328;
   1:L PR[91] R[100]mm/sec CNT100;
   1:  PR[91,1] = PR[90,1] + -15.267;
   1:  PR[91,2] = PR[90,2] + -24.448;
   1:  PR[91,3] = PR[90,3] + 73.351;
   1:L PR[91] R[100]mm/sec CNT100;
   1:  PR[91,1] = PR[90,1] + -12.819;
   1:  PR[91,2] = PR[90,2] + -24.115;
   1:  PR[91,3] = PR[90,3] + 73.354;
   1:L PR[91] R[100]mm/sec CNT100;
   1:  PR[91,1] = PR[90,1] + -9.318;
   1:  PR[91,2] = PR[90,2] + -24.934;
   1:  PR[91,3] = PR[90,3] + 73.363;
   1:L PR[91] R[100]mm/sec CNT100;
   1:  PR[91,1] = PR[90,1] + -4.080;
   1:  PR[91,2] = PR[90,2] + -25.439;
   1:  PR[91,3] = PR[90,3] + 73.376;
   1:L PR[91] R[100]mm/sec CNT100;
   1:  PR[91,1] = PR[90,1] + -3.098;
   1:  PR[91,2] = PR[90,2] + -25.518;
   1:  PR[91,3] = PR[90,3] + 73.396;
   1:L PR[91] R[100]mm/sec CNT100;
   1:  PR[91,1] = PR[90,1] + -0.263;
   1:  PR[91,2] = PR[90,2] + -25.271;
   1:  PR[91,3] = PR[90,3] + 73.400;
   1:L PR[91] R[100]mm/sec CNT100;
   1:  PR[91,1] = PR[90,1] + 3.076;
   1:  PR[91,2] = PR[90,2] + -25.040;
   1:  PR[91,3] = PR[90,3] + 73.410;
   1:L PR[91] R[100]mm/sec CNT100;
   1:  PR[91,1] = PR[90,1] + 3.877;
   1:  PR[91,2] = PR[90,2] + -24.945;
   1:  PR[91,3] = PR[90,3] + 73.423;
   1:L PR[91] R[100]mm/sec CNT100;
   1:  PR[91,1] = PR[90,1] + 3.950;
   1:  PR[91,2] = PR[90,2] + -24.930;
   1:  PR[91,3] = PR[90,3] + 73.426;
   1:L PR[91] R[100]mm/sec CNT100;
   1:  PR[91,1] = PR[90,1] + 8.541;
   1:  PR[91,2] = PR[90,2] + -23.752;
   1:L PR[91] R[100]mm/sec CNT100;
   1:  PR[91,1] = PR[90,1] + 10.937;
   1:  PR[91,2] = PR[90,2] + -24.852;
   1:  PR[91,3] = PR[90,3] + 73.444;
   1:L PR[91] R[100]mm/sec CNT100;
   1:  PR[91,1] = PR[90,1] + 12.957;
   1:  PR[91,2] = PR[90,2] + -25.403;
   1:  PR[91,3] = PR[90,3] + 73.454;
   1:L PR[91] R[100]mm/sec CNT100;
   1:  PR[91,1] = PR[90,1] + 16.946;
   1:  PR[91,2] = PR[90,2] + -26.263;
   1:  PR[91,3] = PR[90,3] + 73.462;
   1:L PR[91] R[100]mm/sec CNT100;
   1:  PR[91,1] = PR[90,1] + 19.390;
   1:  PR[91,2] = PR[90,2] + -26.362;
   1:  PR[91,3] = PR[90,3] + 73.477;
   1:L PR[91] R[100]mm/sec CNT100;
   1:  PR[91,1] = PR[90,1] + 23.020;
   1:  PR[91,2] = PR[90,2] + -26.246;
   1:  PR[91,3] = PR[90,3] + 73.486;
   1:L PR[91] R[100]mm/sec CNT100;
   1:  PR[91,1] = PR[90,1] + 26.166;
   1:  PR[91,2] = PR[90,2] + -25.768;
   1:  PR[91,3] = PR[90,3] + 73.500;
   1:L PR[91] R[100]mm/sec CNT100;
   1:  PR[91,1] = PR[90,1] + 30.789;
   1:  PR[91,2] = PR[90,2] + -26.975;
   1:  PR[91,3] = PR[90,3] + 73.512;
   1:L PR[91] R[100]mm/sec CNT100;
   1:  PR[91,1] = PR[90,1] + 31.389;
   1:  PR[91,2] = PR[90,2] + -27.119;
   1:  PR[91,3] = PR[90,3] + 73.530;
   1:L PR[91] R[100]mm/sec CNT100;
   1:  PR[91,1] = PR[90,1] + 31.607;
   1:  PR[91,2] = PR[90,2] + -27.149;
   1:  PR[91,3] = PR[90,3] + 73.532;
   1:L PR[91] R[100]mm/sec CNT100;
   1:  PR[91,1] = PR[90,1] + 36.451;
   1:  PR[91,2] = PR[90,2] + -27.543;
   1:  PR[91,3] = PR[90,3] + 73.533;
   1:L PR[91] R[100]mm/sec CNT100;
   1:  PR[91,1] = PR[90,1] + 39.115;
   1:  PR[91,2] = PR[90,2] + -27.498;
   1:  PR[91,3] = PR[90,3] + 73.551;
   1:L PR[91] R[100]mm/sec CNT100;
   1:  PR[91,1] = PR[90,1] + 41.086;
   1:  PR[91,2] = PR[90,2] + -27.346;
   1:  PR[91,3] = PR[90,3] + 73.561;
   1:L PR[91] R[100]mm/sec CNT100;
   1:  PR[91,1] = PR[90,1] + 44.077;
   1:  PR[91,2] = PR[90,2] + -26.831;
   1:  PR[91,3] = PR[90,3] + 73.569;
   1:L PR[91] R[100]mm/sec CNT100;
   1:  PR[91,1] = PR[90,1] + 45.841;
   1:  PR[91,2] = PR[90,2] + -26.594;
   1:  PR[91,3] = PR[90,3] + 73.580;
   1:L PR[91] R[100]mm/sec CNT100;
   1:  PR[91,1] = PR[90,1] + 47.415;
   1:  PR[91,2] = PR[90,2] + -26.203;
   1:  PR[91,3] = PR[90,3] + 73.587;
   1:L PR[91] R[100]mm/sec CNT100;
   1:  PR[91,1] = PR[90,1] + 50.701;
   1:  PR[91,2] = PR[90,2] + -25.316;
   1:  PR[91,3] = PR[90,3] + 73.593;
   1:L PR[91] R[100]mm/sec CNT100;
   1:  PR[91,1] = PR[90,1] + 53.247;
   1:  PR[91,2] = PR[90,2] + -24.327;
   1:  PR[91,3] = PR[90,3] + 73.605;
   1:L PR[91] R[100]mm/sec CNT100;
   1:  PR[91,1] = PR[90,1] + 55.044;
   1:  PR[91,2] = PR[90,2] + -23.740;
   1:  PR[91,3] = PR[90,3] + 73.616;
   1:L PR[91] R[100]mm/sec CNT100;
   1:  PR[91,1] = PR[90,1] + 59.326;
   1:  PR[91,2] = PR[90,2] + -21.797;
   1:  PR[91,3] = PR[90,3] + 73.623;
   1:L PR[91] R[100]mm/sec CNT100;
   1:  PR[91,1] = PR[90,1] + 63.257;
   1:  PR[91,2] = PR[90,2] + -19.293;
   1:  PR[91,3] = PR[90,3] + 73.640;
   1:L PR[91] R[100]mm/sec CNT100;
   1:  PR[91,1] = PR[90,1] + 64.999;
   1:  PR[91,2] = PR[90,2] + -17.857;
   1:  PR[91,3] = PR[90,3] + 73.658;
   1:L PR[91] R[100]mm/sec CNT100;
   1:  PR[91,1] = PR[90,1] + 67.258;
   1:  PR[91,2] = PR[90,2] + -15.869;
   1:  PR[91,3] = PR[90,3] + 73.666;
   1:L PR[91] R[100]mm/sec CNT100;
   1:  PR[91,1] = PR[90,1] + 69.969;
   1:  PR[91,2] = PR[90,2] + -12.422;
   1:  PR[91,3] = PR[90,3] + 73.678;
   1:L PR[91] R[100]mm/sec CNT100;
   1:  PR[91,1] = PR[90,1] + 70.849;
   1:  PR[91,2] = PR[90,2] + -11.330;
   1:  PR[91,3] = PR[90,3] + 73.694;
   1:L PR[91] R[100]mm/sec CNT100;
   1:  PR[91,1] = PR[90,1] + 71.207;
   1:  PR[91,2] = PR[90,2] + -10.686;
   1:  PR[91,3] = PR[90,3] + 73.699;
   1:L PR[91] R[100]mm/sec CNT100;
   1:  PR[91,1] = PR[90,1] + 73.223;
   1:  PR[91,2] = PR[90,2] + -6.082;
   1:  PR[91,3] = PR[90,3] + 73.702;
   1:L PR[91] R[100]mm/sec CNT100;
   1:  PR[91,1] = PR[90,1] + 73.252;
   1:  PR[91,2] = PR[90,2] + -5.992;
   1:  PR[91,3] = PR[90,3] + 73.721;
   1:L PR[91] R[100]mm/sec CNT100;
   1:  PR[91,1] = PR[90,1] + 74.000;
   1:  PR[91,2] = PR[90,2] + -0.732;
   1:L PR[91] R[100]mm/sec CNT100;
   1:  PR[91,1] = PR[90,1] + 73.258;
   1:  PR[91,2] = PR[90,2] + 4.411;
   1:  PR[91,3] = PR[90,3] + 73.741;
   1:L PR[91] R[100]mm/sec CNT100;
   1:  PR[91,1] = PR[90,1] + 73.242;
   1:  PR[91,2] = PR[90,2] + 4.566;
   1:  PR[91,3] = PR[90,3] + 73.761;
   1:L PR[91] R[100]mm/sec CNT100;
   1:  PR[91,1] = PR[90,1] + 73.224;
   1:  PR[91,2] = PR[90,2] + 4.620;
   1:L PR[91] R[100]mm/sec CNT100;
   1:  PR[91,1] = PR[90,1] + 71.210;
   1:  PR[91,2] = PR[90,2] + 9.223;
   1:  PR[91,3] = PR[90,3] + 73.762;
   1:L PR[91] R[100]mm/sec CNT100;
   1:  PR[91,1] = PR[90,1] + 70.845;
   1:  PR[91,2] = PR[90,2] + 9.879;
   1:  PR[91,3] = PR[90,3] + 73.780;
   1:L PR[91] R[100]mm/sec CNT100;
   1:  PR[91,1] = PR[90,1] + 68.354;
   1:  PR[91,2] = PR[90,2] + 13.068;
   1:  PR[91,3] = PR[90,3] + 73.783;
   1:L PR[91] R[100]mm/sec CNT100;
   1:  PR[91,1] = PR[90,1] + 67.275;
   1:  PR[91,2] = PR[90,2] + 14.395;
   1:  PR[91,3] = PR[90,3] + 73.798;
   1:L PR[91] R[100]mm/sec CNT100;
   1:  PR[91,1] = PR[90,1] + 65.003;
   1:  PR[91,2] = PR[90,2] + 16.394;
   1:  PR[91,3] = PR[90,3] + 73.805;
   1:L PR[91] R[100]mm/sec CNT100;
   1:  PR[91,1] = PR[90,1] + 63.260;
   1:  PR[91,2] = PR[90,2] + 17.832;
   1:  PR[91,3] = PR[90,3] + 73.816;
   1:L PR[91] R[100]mm/sec CNT100;
   1:  PR[91,1] = PR[90,1] + 59.326;
   1:  PR[91,2] = PR[90,2] + 20.338;
   1:  PR[91,3] = PR[90,3] + 73.825;
   1:L PR[91] R[100]mm/sec CNT100;
   1:  PR[91,1] = PR[90,1] + 55.044;
   1:  PR[91,2] = PR[90,2] + 22.281;
   1:  PR[91,3] = PR[90,3] + 73.842;
   1:L PR[91] R[100]mm/sec CNT100;
   1:  PR[91,1] = PR[90,1] + 53.247;
   1:  PR[91,2] = PR[90,2] + 22.869;
   1:  PR[91,3] = PR[90,3] + 73.860;
   1:L PR[91] R[100]mm/sec CNT100;
   1:  PR[91,1] = PR[90,1] + 50.701;
   1:  PR[91,2] = PR[90,2] + 23.857;
   1:  PR[91,3] = PR[90,3] + 73.867;
   1:L PR[91] R[100]mm/sec CNT100;
   1:  PR[91,1] = PR[90,1] + 47.416;
   1:  PR[91,2] = PR[90,2] + 24.744;
   1:  PR[91,3] = PR[90,3] + 73.877;
   1:L PR[91] R[100]mm/sec CNT100;
   1:  PR[91,1] = PR[90,1] + 45.841;
   1:  PR[91,2] = PR[90,2] + 25.135;
   1:  PR[91,3] = PR[90,3] + 73.890;
   1:L PR[91] R[100]mm/sec CNT100;
   1:  PR[91,1] = PR[90,1] + 44.077;
   1:  PR[91,2] = PR[90,2] + 25.372;
   1:  PR[91,3] = PR[90,3] + 73.896;
   1:L PR[91] R[100]mm/sec CNT100;
   1:  PR[91,1] = PR[90,1] + 41.086;
   1:  PR[91,2] = PR[90,2] + 25.887;
   1:  PR[91,3] = PR[90,3] + 73.903;
   1:L PR[91] R[100]mm/sec CNT100;
   1:  PR[91,1] = PR[90,1] + 39.115;
   1:  PR[91,2] = PR[90,2] + 26.039;
   1:  PR[91,3] = PR[90,3] + 73.914;
   1:L PR[91] R[100]mm/sec CNT100;
   1:  PR[91,1] = PR[90,1] + 36.451;
   1:  PR[91,2] = PR[90,2] + 26.084;
   1:  PR[91,3] = PR[90,3] + 73.921;
   1:L PR[91] R[100]mm/sec CNT100;
   1:  PR[91,1] = PR[90,1] + 31.607;
   1:  PR[91,2] = PR[90,2] + 25.690;
   1:  PR[91,3] = PR[90,3] + 73.931;
   1:L PR[91] R[100]mm/sec CNT100;
   1:  PR[91,1] = PR[90,1] + 31.390;
   1:  PR[91,2] = PR[90,2] + 25.660;
   1:  PR[91,3] = PR[90,3] + 73.950;
   1:L PR[91] R[100]mm/sec CNT100;
   1:  PR[91,1] = PR[90,1] + 30.789;
   1:  PR[91,2] = PR[90,2] + 25.516;
   1:L PR[91] R[100]mm/sec CNT100;
   1:  PR[91,1] = PR[90,1] + 26.166;
   1:  PR[91,2] = PR[90,2] + 24.310;
   1:  PR[91,3] = PR[90,3] + 73.953;
   1:L PR[91] R[100]mm/sec CNT100;
   1:  PR[91,1] = PR[90,1] + 23.020;
   1:  PR[91,2] = PR[90,2] + 24.787;
   1:  PR[91,3] = PR[90,3] + 73.971;
   1:L PR[91] R[100]mm/sec CNT100;
   1:  PR[91,1] = PR[90,1] + 19.389;
   1:  PR[91,2] = PR[90,2] + 24.904;
   1:  PR[91,3] = PR[90,3] + 73.983;
   1:L PR[91] R[100]mm/sec CNT100;
   1:  PR[91,1] = PR[90,1] + 16.945;
   1:  PR[91,2] = PR[90,2] + 24.804;
   1:  PR[91,3] = PR[90,3] + 73.996;
   1:L PR[91] R[100]mm/sec CNT100;
   1:  PR[91,1] = PR[90,1] + 12.957;
   1:  PR[91,2] = PR[90,2] + 23.944;
   1:  PR[91,3] = PR[90,3] + 74.005;
   1:L PR[91] R[100]mm/sec CNT100;
   1:  PR[91,1] = PR[90,1] + 10.936;
   1:  PR[91,2] = PR[90,2] + 23.393;
   1:  PR[91,3] = PR[90,3] + 74.021;
   1:L PR[91] R[100]mm/sec CNT100;
   1:  PR[91,1] = PR[90,1] + 8.540;
   1:  PR[91,2] = PR[90,2] + 22.294;
   1:  PR[91,3] = PR[90,3] + 74.029;
   1:L PR[91] R[100]mm/sec CNT100;
   1:  PR[91,1] = PR[90,1] + 3.990;
   1:  PR[91,2] = PR[90,2] + 23.465;
   1:  PR[91,3] = PR[90,3] + 74.038;
   1:L PR[91] R[100]mm/sec CNT100;
   1:  PR[91,1] = PR[90,1] + 3.918;
   1:  PR[91,2] = PR[90,2] + 23.480;
   1:  PR[91,3] = PR[90,3] + 74.056;
   1:L PR[91] R[100]mm/sec CNT100;
   1:  PR[91,1] = PR[90,1] + 3.110;
   1:  PR[91,2] = PR[90,2] + 23.575;
   1:L PR[91] R[100]mm/sec CNT100;
   1:  PR[91,1] = PR[90,1] + -0.265;
   1:  PR[91,2] = PR[90,2] + 23.811;
   1:  PR[91,3] = PR[90,3] + 74.059;
   1:L PR[91] R[100]mm/sec CNT100;
   1:  PR[91,1] = PR[90,1] + -3.075;
   1:  PR[91,2] = PR[90,2] + 24.060;
   1:  PR[91,3] = PR[90,3] + 74.072;
   1:L PR[91] R[100]mm/sec CNT100;
   1:  PR[91,1] = PR[90,1] + -4.049;
   1:  PR[91,2] = PR[90,2] + 23.981;
   1:  PR[91,3] = PR[90,3] + 74.083;
   1:L PR[91] R[100]mm/sec CNT100;
   1:  PR[91,1] = PR[90,1] + -9.316;
   1:  PR[91,2] = PR[90,2] + 23.475;
   1:  PR[91,3] = PR[90,3] + 74.086;
   1:L PR[91] R[100]mm/sec CNT100;
   1:  PR[91,1] = PR[90,1] + -12.817;
   1:  PR[91,2] = PR[90,2] + 22.655;
   1:  PR[91,3] = PR[90,3] + 74.106;
   1:L PR[91] R[100]mm/sec CNT100;
   1:  PR[91,1] = PR[90,1] + -15.342;
   1:  PR[91,2] = PR[90,2] + 22.999;
   1:  PR[91,3] = PR[90,3] + 74.120;
   1:L PR[91] R[100]mm/sec CNT100;
   1:  PR[91,1] = PR[90,1] + -20.795;
   1:  PR[91,2] = PR[90,2] + 23.595;
   1:  PR[91,3] = PR[90,3] + 74.129;
   1:L PR[91] R[100]mm/sec CNT100;
   1:  PR[91,1] = PR[90,1] + -22.236;
   1:  PR[91,2] = PR[90,2] + 23.727;
   1:  PR[91,3] = PR[90,3] + 74.150;
   1:L PR[91] R[100]mm/sec CNT100;
   1:  PR[91,1] = PR[90,1] + -27.838;
   1:  PR[91,2] = PR[90,2] + 23.938;
   1:  PR[91,3] = PR[90,3] + 74.155;
   1:L PR[91] R[100]mm/sec CNT100;
   1:  PR[91,1] = PR[90,1] + -33.003;
   1:  PR[91,2] = PR[90,2] + 24.087;
   1:  PR[91,3] = PR[90,3] + 74.176;
   1:L PR[91] R[100]mm/sec CNT100;
   1:  PR[91,1] = PR[90,1] + -35.299;
   1:  PR[91,2] = PR[90,2] + 24.022;
   1:  PR[91,3] = PR[90,3] + 74.196;
   1:L PR[91] R[100]mm/sec CNT100;
   1:  PR[91,1] = PR[90,1] + -37.275;
   1:  PR[91,2] = PR[90,2] + 23.854;
   1:  PR[91,3] = PR[90,3] + 74.204;
   1:L PR[91] R[100]mm/sec CNT100;
   1:  PR[91,1] = PR[90,1] + -42.440;
   1:  PR[91,2] = PR[90,2] + 23.513;
   1:  PR[91,3] = PR[90,3] + 74.212;
   1:L PR[91] R[100]mm/sec CNT100;
   1:  PR[91,1] = PR[90,1] + -49.331;
   1:  PR[91,2] = PR[90,2] + 22.340;
   1:  PR[91,3] = PR[90,3] + 74.231;
   1:L PR[91] R[100]mm/sec CNT100;
   1:  PR[91,1] = PR[90,1] + -50.017;
   1:  PR[91,2] = PR[90,2] + 22.199;
   1:  PR[91,3] = PR[90,3] + 74.257;
   1:L PR[91] R[100]mm/sec CNT100;
   1:  PR[91,1] = PR[90,1] + -54.206;
   1:  PR[91,2] = PR[90,2] + 20.829;
   1:  PR[91,3] = PR[90,3] + 74.260;
   1:L PR[91] R[100]mm/sec CNT100;
   1:  PR[91,1] = PR[90,1] + -57.892;
   1:  PR[91,2] = PR[90,2] + 19.487;
   1:  PR[91,3] = PR[90,3] + 74.276;
   1:L PR[91] R[100]mm/sec CNT100;
   1:  PR[91,1] = PR[90,1] + -58.805;
   1:  PR[91,2] = PR[90,2] + 19.009;
   1:  PR[91,3] = PR[90,3] + 74.291;
   1:L PR[91] R[100]mm/sec CNT100;
   1:  PR[91] = PR[90];
   1:  PR[91,1] = PR[90,1] + -62.230;
   1:  PR[91,2] = PR[90,2] + 16.537;
   1:  PR[91,3] = PR[90,3] + 75.595;
   1:L PR[91] R[100]mm/sec CNT100;
   1:  PR[91,1] = PR[90,1] + -62.554;
   1:  PR[91,2] = PR[90,2] + 16.339;
   1:  PR[91,3] = PR[90,3] + 74.312;
   1:L PR[91] R[100]mm/sec CNT100;
   1:  PR[91,1] = PR[90,1] + -66.769;
   1:  PR[91,2] = PR[90,2] + 12.501;
   1:  PR[91,3] = PR[90,3] + 74.314;
   1:L PR[91] R[100]mm/sec CNT100;
   1:  PR[91,1] = PR[90,1] + -69.779;
   1:  PR[91,2] = PR[90,2] + 8.278;
   1:  PR[91,3] = PR[90,3] + 74.335;
   1:L PR[91] R[100]mm/sec CNT100;
   1:  PR[91,1] = PR[90,1] + -71.575;
   1:  PR[91,2] = PR[90,2] + 3.825;
   1:  PR[91,3] = PR[90,3] + 74.355;
   1:L PR[91] R[100]mm/sec CNT100;
   1:  PR[91,1] = PR[90,1] + -71.976;
   1:  PR[91,2] = PR[90,2] + 0.761;
   1:  PR[91,3] = PR[90,3] + 74.373;
   1:L PR[91] R[100]mm/sec CNT100;
   1:  PR[91,1] = PR[90,1] + -72.233;
   1:  PR[91,2] = PR[90,2] + -0.698;
   1:  PR[91,3] = PR[90,3] + 74.385;
   1:L PR[91] R[100]mm/sec CNT100;
   1:  PR[91,1] = PR[90,1] + -71.979;
   1:  PR[91,2] = PR[90,2] + -1.925;
   1:  PR[91,3] = PR[90,3] + 74.391;
   1:L PR[91] R[100]mm/sec CNT100;
   1:  PR[91,1] = PR[90,1] + -71.526;
   1:  PR[91,2] = PR[90,2] + -5.441;
   1:  PR[91,3] = PR[90,3] + 74.395;
   1:L PR[91] R[100]mm/sec CNT100;
   1:  PR[91,1] = PR[90,1] + -69.959;
   1:  PR[91,2] = PR[90,2] + -9.346;
   1:  PR[91,3] = PR[90,3] + 74.409;
   1:L PR[91] R[100]mm/sec CNT100;
   1:  PR[91,1] = PR[90,1] + -69.692;
   1:  PR[91,2] = PR[90,2] + -10.003;
   1:  PR[91,3] = PR[90,3] + 74.425;
   1:L PR[91] R[100]mm/sec CNT100;
   1:  PR[91,1] = PR[90,1] + -66.856;
   1:  PR[91,2] = PR[90,2] + -13.988;
   1:  PR[91,3] = PR[90,3] + 74.428;
   1:L PR[91] R[100]mm/sec CNT100;
   1:  PR[91,1] = PR[90,1] + -66.676;
   1:  PR[91,2] = PR[90,2] + -14.218;
   1:  PR[91,3] = PR[90,3] + 74.446;
   1:L PR[91] R[100]mm/sec CNT100;
   1:  PR[91,1] = PR[90,1] + -62.353;
   1:  PR[91,2] = PR[90,2] + -17.822;
   1:  PR[91,3] = PR[90,3] + 74.447;
   1:L PR[91] R[100]mm/sec CNT100;
   1:  PR[91,1] = PR[90,1] + -60.340;
   1:  PR[91,2] = PR[90,2] + -19.056;
   1:  PR[91,3] = PR[90,3] + 74.469;
   1:L PR[91] R[100]mm/sec CNT100;
   1:  PR[91,1] = PR[90,1] + -57.328;
   1:  PR[91,2] = PR[90,2] + -20.734;
   1:  PR[91,3] = PR[90,3] + 74.477;
   1:L PR[91] R[100]mm/sec CNT100;
   1:  PR[91,1] = PR[90,1] + -51.882;
   1:  PR[91,2] = PR[90,2] + -22.951;
   1:  PR[91,3] = PR[90,3] + 74.491;
   1:L PR[91] R[100]mm/sec CNT100;
   1:  PR[91,1] = PR[90,1] + -46.501;
   1:  PR[91,2] = PR[90,2] + -24.192;
   1:  PR[91,3] = PR[90,3] + 74.513;
   1:L PR[91] R[100]mm/sec CNT100;
   1:  PR[91,1] = PR[90,1] + -42.429;
   1:  PR[91,2] = PR[90,2] + -24.992;
   1:  PR[91,3] = PR[90,3] + 74.534;
   1:L PR[91] R[100]mm/sec CNT100;
   1:  PR[91,1] = PR[90,1] + -41.016;
   1:  PR[91,2] = PR[90,2] + -25.140;
   1:  PR[91,3] = PR[90,3] + 74.550;
   1:L PR[91] R[100]mm/sec CNT100;
   1:  PR[91,1] = PR[90,1] + -39.295;
   1:  PR[91,2] = PR[90,2] + -25.255;
   1:  PR[91,3] = PR[90,3] + 74.555;
   1:L PR[91] R[100]mm/sec CNT100;
   1:  PR[91,1] = PR[90,1] + -34.170;
   1:  PR[91,2] = PR[90,2] + -25.663;
   1:  PR[91,3] = PR[90,3] + 74.561;
   1:L PR[91] R[100]mm/sec CNT100;
   1:  PR[91,1] = PR[90,1] + -29.360;
   1:  PR[91,2] = PR[90,2] + -25.808;
   1:  PR[91,3] = PR[90,3] + 74.581;
   1:L PR[91] R[100]mm/sec CNT100;
   1:  PR[91,1] = PR[90,1] + -19.571;
   1:  PR[91,2] = PR[90,2] + -25.445;
   1:  PR[91,3] = PR[90,3] + 74.599;
   1:L PR[91] R[100]mm/sec CNT100;
   1:  PR[91,1] = PR[90,1] + -19.341;
   1:  PR[91,2] = PR[90,2] + -25.428;
   1:  PR[91,3] = PR[90,3] + 74.636;
   1:L PR[91] R[100]mm/sec CNT100;
   1:  PR[91,1] = PR[90,1] + -13.828;
   1:  PR[91,2] = PR[90,2] + -24.802;
   1:  PR[91,3] = PR[90,3] + 74.637;
   1:L PR[91] R[100]mm/sec CNT100;
   1:  PR[91,1] = PR[90,1] + -13.051;
   1:  PR[91,2] = PR[90,2] + -24.776;
   1:  PR[91,3] = PR[90,3] + 74.658;
   1:L PR[91] R[100]mm/sec CNT100;
   1:  PR[91,1] = PR[90,1] + -11.210;
   1:  PR[91,2] = PR[90,2] + -24.526;
   1:  PR[91,3] = PR[90,3] + 74.661;
   1:L PR[91] R[100]mm/sec CNT100;
   1:  PR[91,1] = PR[90,1] + -8.621;
   1:  PR[91,2] = PR[90,2] + -25.132;
   1:  PR[91,3] = PR[90,3] + 74.668;
   1:L PR[91] R[100]mm/sec CNT100;
   1:  PR[91,1] = PR[90,1] + -2.308;
   1:  PR[91,2] = PR[90,2] + -25.739;
   1:  PR[91,3] = PR[90,3] + 74.678;
   1:L PR[91] R[100]mm/sec CNT100;
   1:  PR[91,1] = PR[90,1] + 3.588;
   1:  PR[91,2] = PR[90,2] + -25.327;
   1:  PR[91,3] = PR[90,3] + 74.702;
   1:L PR[91] R[100]mm/sec CNT100;
   1:  PR[91,1] = PR[90,1] + 5.072;
   1:  PR[91,2] = PR[90,2] + -25.151;
   1:  PR[91,3] = PR[90,3] + 74.725;
   1:L PR[91] R[100]mm/sec CNT100;
   1:  PR[91,1] = PR[90,1] + 5.294;
   1:  PR[91,2] = PR[90,2] + -25.106;
   1:  PR[91,3] = PR[90,3] + 74.730;
   1:L PR[91] R[100]mm/sec CNT100;
   1:  PR[91,1] = PR[90,1] + 8.887;
   1:  PR[91,2] = PR[90,2] + -24.184;
   1:  PR[91,3] = PR[90,3] + 74.731;
   1:L PR[91] R[100]mm/sec CNT100;
   1:  PR[91,1] = PR[90,1] + 10.803;
   1:  PR[91,2] = PR[90,2] + -25.064;
   1:  PR[91,3] = PR[90,3] + 74.745;
   1:L PR[91] R[100]mm/sec CNT100;
   1:  PR[91,1] = PR[90,1] + 12.260;
   1:  PR[91,2] = PR[90,2] + -25.461;
   1:  PR[91,3] = PR[90,3] + 74.753;
   1:L PR[91] R[100]mm/sec CNT100;
   1:  PR[91,1] = PR[90,1] + 16.908;
   1:  PR[91,2] = PR[90,2] + -26.464;
   1:  PR[91,3] = PR[90,3] + 74.759;
   1:L PR[91] R[100]mm/sec CNT100;
   1:  PR[91,1] = PR[90,1] + 18.784;
   1:  PR[91,2] = PR[90,2] + -26.540;
   1:  PR[91,3] = PR[90,3] + 74.777;
   1:L PR[91] R[100]mm/sec CNT100;
   1:  PR[91,1] = PR[90,1] + 23.071;
   1:  PR[91,2] = PR[90,2] + -26.402;
   1:  PR[91,3] = PR[90,3] + 74.784;
   1:L PR[91] R[100]mm/sec CNT100;
   1:  PR[91,1] = PR[90,1] + 25.698;
   1:  PR[91,2] = PR[90,2] + -26.004;
   1:  PR[91,3] = PR[90,3] + 74.800;
   1:L PR[91] R[100]mm/sec CNT100;
   1:  PR[91,1] = PR[90,1] + 30.362;
   1:  PR[91,2] = PR[90,2] + -27.222;
   1:  PR[91,3] = PR[90,3] + 74.811;
   1:L PR[91] R[100]mm/sec CNT100;
   1:  PR[91,1] = PR[90,1] + 30.917;
   1:  PR[91,2] = PR[90,2] + -27.349;
   1:  PR[91,3] = PR[90,3] + 74.829;
   1:L PR[91] R[100]mm/sec CNT100;
   1:  PR[91,1] = PR[90,1] + 36.092;
   1:  PR[91,2] = PR[90,2] + -27.767;
   1:  PR[91,3] = PR[90,3] + 74.831;
   1:L PR[91] R[100]mm/sec CNT100;
   1:  PR[91,1] = PR[90,1] + 37.562;
   1:  PR[91,2] = PR[90,2] + -27.742;
   1:  PR[91,3] = PR[90,3] + 74.851;
   1:L PR[91] R[100]mm/sec CNT100;
   1:  PR[91,1] = PR[90,1] + 40.843;
   1:  PR[91,2] = PR[90,2] + -27.489;
   1:  PR[91,3] = PR[90,3] + 74.856;
   1:L PR[91] R[100]mm/sec CNT100;
   1:  PR[91,1] = PR[90,1] + 44.859;
   1:  PR[91,2] = PR[90,2] + -26.798;
   1:  PR[91,3] = PR[90,3] + 74.869;
   1:L PR[91] R[100]mm/sec CNT100;
   1:  PR[91,1] = PR[90,1] + 45.035;
   1:  PR[91,2] = PR[90,2] + -26.755;
   1:  PR[91,3] = PR[90,3] + 74.884;
   1:L PR[91] R[100]mm/sec CNT100;
   1:  PR[91,1] = PR[90,1] + 45.439;
   1:  PR[91,2] = PR[90,2] + -26.620;
   1:  PR[91,3] = PR[90,3] + 74.885;
   1:L PR[91] R[100]mm/sec CNT100;
   1:  PR[91,1] = PR[90,1] + 50.066;
   1:  PR[91,2] = PR[90,2] + -25.370;
   1:  PR[91,3] = PR[90,3] + 74.886;
   1:L PR[91] R[100]mm/sec CNT100;
   1:  PR[91,1] = PR[90,1] + 54.222;
   1:  PR[91,2] = PR[90,2] + -23.752;
   1:  PR[91,3] = PR[90,3] + 74.905;
   1:L PR[91] R[100]mm/sec CNT100;
   1:  PR[91,1] = PR[90,1] + 58.483;
   1:  PR[91,2] = PR[90,2] + -21.746;
   1:  PR[91,3] = PR[90,3] + 74.922;
   1:L PR[91] R[100]mm/sec CNT100;
   1:  PR[91,1] = PR[90,1] + 60.714;
   1:  PR[91,2] = PR[90,2] + -20.361;
   1:  PR[91,3] = PR[90,3] + 74.939;
   1:L PR[91] R[100]mm/sec CNT100;
   1:  PR[91,1] = PR[90,1] + 62.441;
   1:  PR[91,2] = PR[90,2] + -19.259;
   1:  PR[91,3] = PR[90,3] + 74.949;
   1:L PR[91] R[100]mm/sec CNT100;
   1:  PR[91,1] = PR[90,1] + 63.212;
   1:  PR[91,2] = PR[90,2] + -18.624;
   1:  PR[91,3] = PR[90,3] + 74.957;
   1:L PR[91] R[100]mm/sec CNT100;
   1:  PR[91,1] = PR[90,1] + 66.249;
   1:  PR[91,2] = PR[90,2] + -15.952;
   1:  PR[91,3] = PR[90,3] + 74.961;
   1:L PR[91] R[100]mm/sec CNT100;
   1:  PR[91,1] = PR[90,1] + 68.196;
   1:  PR[91,2] = PR[90,2] + -13.476;
   1:  PR[91,3] = PR[90,3] + 74.976;
   1:L PR[91] R[100]mm/sec CNT100;
   1:  PR[91,1] = PR[90,1] + 69.716;
   1:  PR[91,2] = PR[90,2] + -11.590;
   1:  PR[91,3] = PR[90,3] + 74.988;
   1:L PR[91] R[100]mm/sec CNT100;
   1:  PR[91,1] = PR[90,1] + 70.392;
   1:  PR[91,2] = PR[90,2] + -10.373;
   1:  PR[91,3] = PR[90,3] + 74.997;
   1:L PR[91] R[100]mm/sec CNT100;
   1:  PR[91,1] = PR[90,1] + 72.069;
   1:  PR[91,2] = PR[90,2] + -6.543;
   1:  PR[91,3] = PR[90,3] + 75.003;
   1:L PR[91] R[100]mm/sec CNT100;
   1:  PR[91,1] = PR[90,1] + 72.303;
   1:  PR[91,2] = PR[90,2] + -5.816;
   1:  PR[91,3] = PR[90,3] + 75.018;
   1:L PR[91] R[100]mm/sec CNT100;
   1:  PR[91,1] = PR[90,1] + 72.956;
   1:  PR[91,2] = PR[90,2] + -1.250;
   1:  PR[91,3] = PR[90,3] + 75.021;
   1:L PR[91] R[100]mm/sec CNT100;
   1:  PR[91,1] = PR[90,1] + 73.007;
   1:  PR[91,2] = PR[90,2] + -0.768;
   1:  PR[91,3] = PR[90,3] + 75.039;
   1:L PR[91] R[100]mm/sec CNT100;
   1:  PR[91,1] = PR[90,1] + 72.370;
   1:  PR[91,2] = PR[90,2] + 3.645;
   1:  PR[91,3] = PR[90,3] + 75.041;
   1:L PR[91] R[100]mm/sec CNT100;
   1:  PR[91,1] = PR[90,1] + 72.292;
   1:  PR[91,2] = PR[90,2] + 4.391;
   1:  PR[91,3] = PR[90,3] + 75.058;
   1:L PR[91] R[100]mm/sec CNT100;
   1:  PR[91,1] = PR[90,1] + 72.070;
   1:  PR[91,2] = PR[90,2] + 5.082;
   1:  PR[91,3] = PR[90,3] + 75.060;
   1:L PR[91] R[100]mm/sec CNT100;
   1:  PR[91,1] = PR[90,1] + 70.395;
   1:  PR[91,2] = PR[90,2] + 8.910;
   1:  PR[91,3] = PR[90,3] + 75.063;
   1:L PR[91] R[100]mm/sec CNT100;
   1:  PR[91,1] = PR[90,1] + 69.711;
   1:  PR[91,2] = PR[90,2] + 10.140;
   1:  PR[91,3] = PR[90,3] + 75.079;
   1:L PR[91] R[100]mm/sec CNT100;
   1:  PR[91,1] = PR[90,1] + 67.727;
   1:  PR[91,2] = PR[90,2] + 12.678;
   1:  PR[91,3] = PR[90,3] + 75.084;
   1:L PR[91] R[100]mm/sec CNT100;
   1:  PR[91,1] = PR[90,1] + 66.264;
   1:  PR[91,2] = PR[90,2] + 14.479;
   1:  PR[91,3] = PR[90,3] + 75.097;
   1:L PR[91] R[100]mm/sec CNT100;
   1:  PR[91,1] = PR[90,1] + 63.214;
   1:  PR[91,2] = PR[90,2] + 17.163;
   1:  PR[91,3] = PR[90,3] + 75.105;
   1:L PR[91] R[100]mm/sec CNT100;
   1:  PR[91,1] = PR[90,1] + 62.442;
   1:  PR[91,2] = PR[90,2] + 17.799;
   1:  PR[91,3] = PR[90,3] + 75.121;
   1:L PR[91] R[100]mm/sec CNT100;
   1:  PR[91,1] = PR[90,1] + 60.714;
   1:  PR[91,2] = PR[90,2] + 18.902;
   1:  PR[91,3] = PR[90,3] + 75.125;
   1:L PR[91] R[100]mm/sec CNT100;
   1:  PR[91,1] = PR[90,1] + 58.483;
   1:  PR[91,2] = PR[90,2] + 20.287;
   1:  PR[91,3] = PR[90,3] + 75.132;
   1:L PR[91] R[100]mm/sec CNT100;
   1:  PR[91,1] = PR[90,1] + 54.222;
   1:  PR[91,2] = PR[90,2] + 22.293;
   1:  PR[91,3] = PR[90,3] + 75.142;
   1:L PR[91] R[100]mm/sec CNT100;
   1:  PR[91,1] = PR[90,1] + 50.066;
   1:  PR[91,2] = PR[90,2] + 23.911;
   1:  PR[91,3] = PR[90,3] + 75.160;
   1:L PR[91] R[100]mm/sec CNT100;
   1:  PR[91,1] = PR[90,1] + 45.439;
   1:  PR[91,2] = PR[90,2] + 25.161;
   1:  PR[91,3] = PR[90,3] + 75.177;
   1:L PR[91] R[100]mm/sec CNT100;
   1:  PR[91,1] = PR[90,1] + 45.035;
   1:  PR[91,2] = PR[90,2] + 25.297;
   1:  PR[91,3] = PR[90,3] + 75.195;
   1:L PR[91] R[100]mm/sec CNT100;
   1:  PR[91,1] = PR[90,1] + 44.859;
   1:  PR[91,2] = PR[90,2] + 25.339;
   1:  PR[91,3] = PR[90,3] + 75.197;
   1:L PR[91] R[100]mm/sec CNT100;
   1:  PR[91,1] = PR[90,1] + 40.843;
   1:  PR[91,2] = PR[90,2] + 26.030;
   1:  PR[91,3] = PR[90,3] + 75.198;
   1:L PR[91] R[100]mm/sec CNT100;
   1:  PR[91,1] = PR[90,1] + 37.562;
   1:  PR[91,2] = PR[90,2] + 26.283;
   1:  PR[91,3] = PR[90,3] + 75.213;
   1:L PR[91] R[100]mm/sec CNT100;
   1:  PR[91,1] = PR[90,1] + 36.092;
   1:  PR[91,2] = PR[90,2] + 26.308;
   1:  PR[91,3] = PR[90,3] + 75.225;
   1:L PR[91] R[100]mm/sec CNT100;
   1:  PR[91,1] = PR[90,1] + 30.917;
   1:  PR[91,2] = PR[90,2] + 25.890;
   1:  PR[91,3] = PR[90,3] + 75.231;
   1:L PR[91] R[100]mm/sec CNT100;
   1:  PR[91,1] = PR[90,1] + 30.362;
   1:  PR[91,2] = PR[90,2] + 25.763;
   1:  PR[91,3] = PR[90,3] + 75.251;
   1:L PR[91] R[100]mm/sec CNT100;
   1:  PR[91,1] = PR[90,1] + 25.698;
   1:  PR[91,2] = PR[90,2] + 24.546;
   1:  PR[91,3] = PR[90,3] + 75.253;
   1:L PR[91] R[100]mm/sec CNT100;
   1:  PR[91,1] = PR[90,1] + 23.070;
   1:  PR[91,2] = PR[90,2] + 24.943;
   1:  PR[91,3] = PR[90,3] + 75.271;
   1:L PR[91] R[100]mm/sec CNT100;
   1:  PR[91,1] = PR[90,1] + 18.784;
   1:  PR[91,2] = PR[90,2] + 25.081;
   1:  PR[91,3] = PR[90,3] + 75.281;
   1:L PR[91] R[100]mm/sec CNT100;
   1:  PR[91,1] = PR[90,1] + 16.908;
   1:  PR[91,2] = PR[90,2] + 25.005;
   1:  PR[91,3] = PR[90,3] + 75.298;
   1:L PR[91] R[100]mm/sec CNT100;
   1:  PR[91,1] = PR[90,1] + 12.259;
   1:  PR[91,2] = PR[90,2] + 24.002;
   1:  PR[91,3] = PR[90,3] + 75.305;
   1:L PR[91] R[100]mm/sec CNT100;
   1:  PR[91,1] = PR[90,1] + 10.802;
   1:  PR[91,2] = PR[90,2] + 23.605;
   1:  PR[91,3] = PR[90,3] + 75.323;
   1:L PR[91] R[100]mm/sec CNT100;
   1:  PR[91,1] = PR[90,1] + 8.886;
   1:  PR[91,2] = PR[90,2] + 22.726;
   1:  PR[91,3] = PR[90,3] + 75.328;
   1:L PR[91] R[100]mm/sec CNT100;
   1:  PR[91,1] = PR[90,1] + 5.324;
   1:  PR[91,2] = PR[90,2] + 23.643;
   1:  PR[91,3] = PR[90,3] + 75.336;
   1:L PR[91] R[100]mm/sec CNT100;
   1:  PR[91,1] = PR[90,1] + 5.104;
   1:  PR[91,2] = PR[90,2] + 23.687;
   1:  PR[91,3] = PR[90,3] + 75.350;
   1:L PR[91] R[100]mm/sec CNT100;
   1:  PR[91,1] = PR[90,1] + 3.617;
   1:  PR[91,2] = PR[90,2] + 23.863;
   1:  PR[91,3] = PR[90,3] + 75.351;
   1:L PR[91] R[100]mm/sec CNT100;
   1:  PR[91,1] = PR[90,1] + -2.282;
   1:  PR[91,2] = PR[90,2] + 24.280;
   1:  PR[91,3] = PR[90,3] + 75.357;
   1:L PR[91] R[100]mm/sec CNT100;
   1:  PR[91,1] = PR[90,1] + -8.620;
   1:  PR[91,2] = PR[90,2] + 23.673;
   1:  PR[91,3] = PR[90,3] + 75.379;
   1:L PR[91] R[100]mm/sec CNT100;
   1:  PR[91,1] = PR[90,1] + -11.209;
   1:  PR[91,2] = PR[90,2] + 23.066;
   1:  PR[91,3] = PR[90,3] + 75.403;
   1:L PR[91] R[100]mm/sec CNT100;
   1:  PR[91,1] = PR[90,1] + -13.126;
   1:  PR[91,2] = PR[90,2] + 23.328;
   1:  PR[91,3] = PR[90,3] + 75.413;
   1:L PR[91] R[100]mm/sec CNT100;
   1:  PR[91,1] = PR[90,1] + -16.975;
   1:  PR[91,2] = PR[90,2] + 23.749;
   1:  PR[91,3] = PR[90,3] + 75.421;
   1:L PR[91] R[100]mm/sec CNT100;
   1:  PR[91,1] = PR[90,1] + -19.485;
   1:  PR[91,2] = PR[90,2] + 23.979;
   1:  PR[91,3] = PR[90,3] + 75.436;
   1:L PR[91] R[100]mm/sec CNT100;
   1:  PR[91,1] = PR[90,1] + -29.474;
   1:  PR[91,2] = PR[90,2] + 24.347;
   1:  PR[91,3] = PR[90,3] + 75.445;
   1:L PR[91] R[100]mm/sec CNT100;
   1:  PR[91,1] = PR[90,1] + -34.147;
   1:  PR[91,2] = PR[90,2] + 24.216;
   1:  PR[91,3] = PR[90,3] + 75.483;
   1:L PR[91] R[100]mm/sec CNT100;
   1:  PR[91,1] = PR[90,1] + -38.113;
   1:  PR[91,2] = PR[90,2] + 23.878;
   1:  PR[91,3] = PR[90,3] + 75.501;
   1:L PR[91] R[100]mm/sec CNT100;
   1:  PR[91,1] = PR[90,1] + -41.302;
   1:  PR[91,2] = PR[90,2] + 23.667;
   1:  PR[91,3] = PR[90,3] + 75.516;
   1:L PR[91] R[100]mm/sec CNT100;
   1:  PR[91,1] = PR[90,1] + -47.543;
   1:  PR[91,2] = PR[90,2] + 22.599;
   1:  PR[91,3] = PR[90,3] + 75.528;
   1:L PR[91] R[100]mm/sec CNT100;
   1:  PR[91,1] = PR[90,1] + -48.481;
   1:  PR[91,2] = PR[90,2] + 22.419;
   1:  PR[91,3] = PR[90,3] + 75.552;
   1:L PR[91] R[100]mm/sec CNT100;
   1:  PR[91,1] = PR[90,1] + -53.662;
   1:  PR[91,2] = PR[90,2] + 20.734;
   1:  PR[91,3] = PR[90,3] + 75.556;
   1:L PR[91] R[100]mm/sec CNT100;
   1:  PR[91,1] = PR[90,1] + -56.367;
   1:  PR[91,2] = PR[90,2] + 19.749;
   1:  PR[91,3] = PR[90,3] + 75.576;
   1:L PR[91] R[100]mm/sec CNT100;
   1:  PR[91,1] = PR[90,1] + -58.214;
   1:  PR[91,2] = PR[90,2] + 18.783;
   1:  PR[91,3] = PR[90,3] + 75.587;
   1:L PR[91] R[100]mm/sec CNT100;
   1:  PR[91] = PR[90];
   1:  PR[91,1] = PR[90,1] + -61.321;
   1:  PR[91,2] = PR[90,2] + 16.488;
   1:  PR[91,3] = PR[90,3] + 76.895;
   1:L PR[91] R[100]mm/sec CNT100;
   1:  PR[91,1] = PR[90,1] + -61.751;
   1:  PR[91,2] = PR[90,2] + 16.148;
   1:  PR[91,3] = PR[90,3] + 75.611;
   1:L PR[91] R[100]mm/sec CNT100;
   1:  PR[91,1] = PR[90,1] + -63.245;
   1:  PR[91,2] = PR[90,2] + 14.908;
   1:  PR[91,3] = PR[90,3] + 75.613;
   1:L PR[91] R[100]mm/sec CNT100;
   1:  PR[91,1] = PR[90,1] + -65.760;
   1:  PR[91,2] = PR[90,2] + 12.618;
   1:  PR[91,3] = PR[90,3] + 75.621;
   1:L PR[91] R[100]mm/sec CNT100;
   1:  PR[91,1] = PR[90,1] + -68.800;
   1:  PR[91,2] = PR[90,2] + 8.357;
   1:  PR[91,3] = PR[90,3] + 75.634;
   1:L PR[91] R[100]mm/sec CNT100;
   1:  PR[91,1] = PR[90,1] + -70.612;
   1:  PR[91,2] = PR[90,2] + 3.865;
   1:  PR[91,3] = PR[90,3] + 75.654;
   1:L PR[91] R[100]mm/sec CNT100;
   1:  PR[91,1] = PR[90,1] + -70.919;
   1:  PR[91,2] = PR[90,2] + 1.527;
   1:  PR[91,3] = PR[90,3] + 75.672;
   1:L PR[91] R[100]mm/sec CNT100;
   1:  PR[91,1] = PR[90,1] + -71.311;
   1:  PR[91,2] = PR[90,2] + -0.699;
   1:  PR[91,3] = PR[90,3] + 75.682;
   1:L PR[91] R[100]mm/sec CNT100;
   1:  PR[91,1] = PR[90,1] + -71.180;
   1:  PR[91,2] = PR[90,2] + -1.329;
   1:  PR[91,3] = PR[90,3] + 75.690;
   1:L PR[91] R[100]mm/sec CNT100;
   1:  PR[91,1] = PR[90,1] + -70.648;
   1:  PR[91,2] = PR[90,2] + -5.468;
   1:  PR[91,3] = PR[90,3] + 75.693;
   1:L PR[91] R[100]mm/sec CNT100;
   1:  PR[91,1] = PR[90,1] + -68.806;
   1:  PR[91,2] = PR[90,2] + -10.057;
   1:  PR[91,3] = PR[90,3] + 75.709;
   1:L PR[91] R[100]mm/sec CNT100;
   1:  PR[91,1] = PR[90,1] + -68.274;
   1:  PR[91,2] = PR[90,2] + -10.806;
   1:  PR[91,3] = PR[90,3] + 75.728;
   1:L PR[91] R[100]mm/sec CNT100;
   1:  PR[91,1] = PR[90,1] + -65.619;
   1:  PR[91,2] = PR[90,2] + -14.212;
   1:  PR[91,3] = PR[90,3] + 75.731;
   1:L PR[91] R[100]mm/sec CNT100;
   1:  PR[91,1] = PR[90,1] + -64.867;
   1:  PR[91,2] = PR[90,2] + -14.891;
   1:  PR[91,3] = PR[90,3] + 75.748;
   1:L PR[91] R[100]mm/sec CNT100;
   1:  PR[91,1] = PR[90,1] + -61.355;
   1:  PR[91,2] = PR[90,2] + -17.818;
   1:  PR[91,3] = PR[90,3] + 75.752;
   1:L PR[91] R[100]mm/sec CNT100;
   1:  PR[91,1] = PR[90,1] + -58.279;
   1:  PR[91,2] = PR[90,2] + -19.704;
   1:  PR[91,3] = PR[90,3] + 75.769;
   1:L PR[91] R[100]mm/sec CNT100;
   1:  PR[91,1] = PR[90,1] + -56.388;
   1:  PR[91,2] = PR[90,2] + -20.757;
   1:  PR[91,3] = PR[90,3] + 75.783;
   1:L PR[91] R[100]mm/sec CNT100;
   1:  PR[91,1] = PR[90,1] + -52.808;
   1:  PR[91,2] = PR[90,2] + -22.216;
   1:  PR[91,3] = PR[90,3] + 75.791;
   1:L PR[91] R[100]mm/sec CNT100;
   1:  PR[91,1] = PR[90,1] + -51.042;
   1:  PR[91,2] = PR[90,2] + -22.876;
   1:  PR[91,3] = PR[90,3] + 75.806;
   1:L PR[91] R[100]mm/sec CNT100;
   1:  PR[91,1] = PR[90,1] + -50.028;
   1:  PR[91,2] = PR[90,2] + -23.222;
   1:  PR[91,3] = PR[90,3] + 75.813;
   1:L PR[91] R[100]mm/sec CNT100;
   1:  PR[91,1] = PR[90,1] + -45.759;
   1:  PR[91,2] = PR[90,2] + -24.206;
   1:  PR[91,3] = PR[90,3] + 75.817;
   1:L PR[91] R[100]mm/sec CNT100;
   1:  PR[91,1] = PR[90,1] + -40.300;
   1:  PR[91,2] = PR[90,2] + -25.279;
   1:  PR[91,3] = PR[90,3] + 75.834;
   1:L PR[91] R[100]mm/sec CNT100;
   1:  PR[91,1] = PR[90,1] + -33.010;
   1:  PR[91,2] = PR[90,2] + -25.861;
   1:  PR[91,3] = PR[90,3] + 75.855;
   1:L PR[91] R[100]mm/sec CNT100;
   1:  PR[91,1] = PR[90,1] + -26.617;
   1:  PR[91,2] = PR[90,2] + -26.061;
   1:  PR[91,3] = PR[90,3] + 75.884;
   1:L PR[91] R[100]mm/sec CNT100;
   1:  PR[91,1] = PR[90,1] + -16.860;
   1:  PR[91,2] = PR[90,2] + -25.700;
   1:  PR[91,3] = PR[90,3] + 75.908;
   1:L PR[91] R[100]mm/sec CNT100;
   1:  PR[91,1] = PR[90,1] + -16.514;
   1:  PR[91,2] = PR[90,2] + -25.675;
   1:  PR[91,3] = PR[90,3] + 75.945;
   1:L PR[91] R[100]mm/sec CNT100;
   1:  PR[91,1] = PR[90,1] + -11.759;
   1:  PR[91,2] = PR[90,2] + -25.135;
   1:  PR[91,3] = PR[90,3] + 75.947;
   1:L PR[91] R[100]mm/sec CNT100;
   1:  PR[91,1] = PR[90,1] + -10.834;
   1:  PR[91,2] = PR[90,2] + -25.105;
   1:  PR[91,3] = PR[90,3] + 75.965;
   1:L PR[91] R[100]mm/sec CNT100;
   1:  PR[91,1] = PR[90,1] + -9.602;
   1:  PR[91,2] = PR[90,2] + -24.937;
   1:  PR[91,3] = PR[90,3] + 75.969;
   1:L PR[91] R[100]mm/sec CNT100;
   1:  PR[91,1] = PR[90,1] + -7.923;
   1:  PR[91,2] = PR[90,2] + -25.330;
   1:  PR[91,3] = PR[90,3] + 75.973;
   1:L PR[91] R[100]mm/sec CNT100;
   1:  PR[91,1] = PR[90,1] + -3.823;
   1:  PR[91,2] = PR[90,2] + -25.725;
   1:  PR[91,3] = PR[90,3] + 75.980;
   1:L PR[91] R[100]mm/sec CNT100;
   1:  PR[91,1] = PR[90,1] + -1.693;
   1:  PR[91,2] = PR[90,2] + -25.951;
   1:  PR[91,3] = PR[90,3] + 75.996;
   1:L PR[91] R[100]mm/sec CNT100;
   1:  PR[91,1] = PR[90,1] + -0.935;
   1:  PR[91,2] = PR[90,2] + -25.962;
   1:  PR[91,3] = PR[90,3] + 76.004;
   1:L PR[91] R[100]mm/sec CNT100;
   1:  PR[91,1] = PR[90,1] + 4.101;
   1:  PR[91,2] = PR[90,2] + -25.614;
   1:  PR[91,3] = PR[90,3] + 76.007;
   1:L PR[91] R[100]mm/sec CNT100;
   1:  PR[91,1] = PR[90,1] + 6.267;
   1:  PR[91,2] = PR[90,2] + -25.357;
   1:  PR[91,3] = PR[90,3] + 76.026;
   1:L PR[91] R[100]mm/sec CNT100;
   1:  PR[91,1] = PR[90,1] + 6.639;
   1:  PR[91,2] = PR[90,2] + -25.282;
   1:  PR[91,3] = PR[90,3] + 76.035;
   1:L PR[91] R[100]mm/sec CNT100;
   1:  PR[91,1] = PR[90,1] + 9.233;
   1:  PR[91,2] = PR[90,2] + -24.616;
   1:  PR[91,3] = PR[90,3] + 76.036;
   1:L PR[91] R[100]mm/sec CNT100;
   1:  PR[91,1] = PR[90,1] + 10.669;
   1:  PR[91,2] = PR[90,2] + -25.276;
   1:  PR[91,3] = PR[90,3] + 76.046;
   1:L PR[91] R[100]mm/sec CNT100;
   1:  PR[91,1] = PR[90,1] + 11.562;
   1:  PR[91,2] = PR[90,2] + -25.519;
   1:  PR[91,3] = PR[90,3] + 76.052;
   1:L PR[91] R[100]mm/sec CNT100;
   1:  PR[91,1] = PR[90,1] + 16.871;
   1:  PR[91,2] = PR[90,2] + -26.664;
   1:  PR[91,3] = PR[90,3] + 76.056;
   1:L PR[91] R[100]mm/sec CNT100;
   1:  PR[91,1] = PR[90,1] + 18.179;
   1:  PR[91,2] = PR[90,2] + -26.717;
   1:  PR[91,3] = PR[90,3] + 76.077;
   1:L PR[91] R[100]mm/sec CNT100;
   1:  PR[91,1] = PR[90,1] + 23.121;
   1:  PR[91,2] = PR[90,2] + -26.558;
   1:  PR[91,3] = PR[90,3] + 76.082;
   1:L PR[91] R[100]mm/sec CNT100;
   1:  PR[91,1] = PR[90,1] + 25.230;
   1:  PR[91,2] = PR[90,2] + -26.240;
   1:  PR[91,3] = PR[90,3] + 76.101;
   1:L PR[91] R[100]mm/sec CNT100;
   1:  PR[91,1] = PR[90,1] + 28.911;
   1:  PR[91,2] = PR[90,2] + -27.201;
   1:  PR[91,3] = PR[90,3] + 76.109;
   1:L PR[91] R[100]mm/sec CNT100;
   1:  PR[91,1] = PR[90,1] + 30.544;
   1:  PR[91,2] = PR[90,2] + -27.575;
   1:  PR[91,3] = PR[90,3] + 76.124;
   1:L PR[91] R[100]mm/sec CNT100;
   1:  PR[91,1] = PR[90,1] + 35.732;
   1:  PR[91,2] = PR[90,2] + -27.991;
   1:  PR[91,3] = PR[90,3] + 76.130;
   1:L PR[91] R[100]mm/sec CNT100;
   1:  PR[91,1] = PR[90,1] + 36.008;
   1:  PR[91,2] = PR[90,2] + -27.986;
   1:  PR[91,3] = PR[90,3] + 76.150;
   1:L PR[91] R[100]mm/sec CNT100;
   1:  PR[91,1] = PR[90,1] + 40.601;
   1:  PR[91,2] = PR[90,2] + -27.632;
   1:  PR[91,3] = PR[90,3] + 76.151;
   1:L PR[91] R[100]mm/sec CNT100;
   1:  PR[91,1] = PR[90,1] + 43.395;
   1:  PR[91,2] = PR[90,2] + -27.151;
   1:  PR[91,3] = PR[90,3] + 76.169;
   1:L PR[91] R[100]mm/sec CNT100;
   1:  PR[91,1] = PR[90,1] + 44.903;
   1:  PR[91,2] = PR[90,2] + -26.790;
   1:  PR[91,3] = PR[90,3] + 76.180;
   1:L PR[91] R[100]mm/sec CNT100;
   1:  PR[91,1] = PR[90,1] + 47.079;
   1:  PR[91,2] = PR[90,2] + -26.059;
   1:  PR[91,3] = PR[90,3] + 76.186;
   1:L PR[91] R[100]mm/sec CNT100;
   1:  PR[91,1] = PR[90,1] + 49.432;
   1:  PR[91,2] = PR[90,2] + -25.424;
   1:  PR[91,3] = PR[90,3] + 76.194;
   1:L PR[91] R[100]mm/sec CNT100;
   1:  PR[91,1] = PR[90,1] + 51.453;
   1:  PR[91,2] = PR[90,2] + -24.639;
   1:  PR[91,3] = PR[90,3] + 76.204;
   1:L PR[91] R[100]mm/sec CNT100;
   1:  PR[91,1] = PR[90,1] + 53.638;
   1:  PR[91,2] = PR[90,2] + -23.715;
   1:  PR[91,3] = PR[90,3] + 76.212;
   1:L PR[91] R[100]mm/sec CNT100;
   1:  PR[91,1] = PR[90,1] + 55.403;
   1:  PR[91,2] = PR[90,2] + -22.742;
   1:  PR[91,3] = PR[90,3] + 76.221;
   1:L PR[91] R[100]mm/sec CNT100;
   1:  PR[91,1] = PR[90,1] + 57.643;
   1:  PR[91,2] = PR[90,2] + -21.692;
   1:  PR[91,3] = PR[90,3] + 76.229;
   1:L PR[91] R[100]mm/sec CNT100;
   1:  PR[91,1] = PR[90,1] + 61.600;
   1:  PR[91,2] = PR[90,2] + -19.230;
   1:  PR[91,3] = PR[90,3] + 76.238;
   1:L PR[91] R[100]mm/sec CNT100;
   1:  PR[91,1] = PR[90,1] + 65.239;
   1:  PR[91,2] = PR[90,2] + -16.034;
   1:  PR[91,3] = PR[90,3] + 76.256;
   1:L PR[91] R[100]mm/sec CNT100;
   1:  PR[91,1] = PR[90,1] + 66.422;
   1:  PR[91,2] = PR[90,2] + -14.530;
   1:  PR[91,3] = PR[90,3] + 76.275;
   1:L PR[91] R[100]mm/sec CNT100;
   1:  PR[91,1] = PR[90,1] + 68.582;
   1:  PR[91,2] = PR[90,2] + -11.849;
   1:  PR[91,3] = PR[90,3] + 76.282;
   1:L PR[91] R[100]mm/sec CNT100;
   1:  PR[91,1] = PR[90,1] + 69.577;
   1:  PR[91,2] = PR[90,2] + -10.060;
   1:  PR[91,3] = PR[90,3] + 76.295;
   1:L PR[91] R[100]mm/sec CNT100;
   1:  PR[91,1] = PR[90,1] + 70.915;
   1:  PR[91,2] = PR[90,2] + -7.005;
   1:  PR[91,3] = PR[90,3] + 76.303;
   1:L PR[91] R[100]mm/sec CNT100;
   1:  PR[91,1] = PR[90,1] + 71.354;
   1:  PR[91,2] = PR[90,2] + -5.640;
   1:  PR[91,3] = PR[90,3] + 76.316;
   1:L PR[91] R[100]mm/sec CNT100;
   1:  PR[91,1] = PR[90,1] + 71.890;
   1:  PR[91,2] = PR[90,2] + -1.894;
   1:  PR[91,3] = PR[90,3] + 76.321;
   1:L PR[91] R[100]mm/sec CNT100;
   1:  PR[91,1] = PR[90,1] + 72.009;
   1:  PR[91,2] = PR[90,2] + -0.768;
   1:  PR[91,3] = PR[90,3] + 76.336;
   1:L PR[91] R[100]mm/sec CNT100;
   1:  PR[91,1] = PR[90,1] + 71.482;
   1:  PR[91,2] = PR[90,2] + 2.880;
   1:  PR[91,3] = PR[90,3] + 76.340;
   1:L PR[91] R[100]mm/sec CNT100;
   1:  PR[91,1] = PR[90,1] + 71.343;
   1:  PR[91,2] = PR[90,2] + 4.216;
   1:  PR[91,3] = PR[90,3] + 76.354;
   1:L PR[91] R[100]mm/sec CNT100;
   1:  PR[91,1] = PR[90,1] + 70.915;
   1:  PR[91,2] = PR[90,2] + 5.544;
   1:  PR[91,3] = PR[90,3] + 76.359;
   1:L PR[91] R[100]mm/sec CNT100;
   1:  PR[91,1] = PR[90,1] + 69.579;
   1:  PR[91,2] = PR[90,2] + 8.598;
   1:  PR[91,3] = PR[90,3] + 76.365;
   1:L PR[91] R[100]mm/sec CNT100;
   1:  PR[91,1] = PR[90,1] + 68.577;
   1:  PR[91,2] = PR[90,2] + 10.401;
   1:  PR[91,3] = PR[90,3] + 76.378;
   1:L PR[91] R[100]mm/sec CNT100;
   1:  PR[91,1] = PR[90,1] + 67.100;
   1:  PR[91,2] = PR[90,2] + 12.290;
   1:  PR[91,3] = PR[90,3] + 76.386;
   1:L PR[91] R[100]mm/sec CNT100;
   1:  PR[91,1] = PR[90,1] + 65.254;
   1:  PR[91,2] = PR[90,2] + 14.562;
   1:  PR[91,3] = PR[90,3] + 76.395;
   1:L PR[91] R[100]mm/sec CNT100;
   1:  PR[91,1] = PR[90,1] + 61.600;
   1:  PR[91,2] = PR[90,2] + 17.771;
   1:  PR[91,3] = PR[90,3] + 76.406;
   1:L PR[91] R[100]mm/sec CNT100;
   1:  PR[91,1] = PR[90,1] + 57.643;
   1:  PR[91,2] = PR[90,2] + 20.234;
   1:  PR[91,3] = PR[90,3] + 76.425;
   1:L PR[91] R[100]mm/sec CNT100;
   1:  PR[91,1] = PR[90,1] + 55.403;
   1:  PR[91,2] = PR[90,2] + 21.284;
   1:  PR[91,3] = PR[90,3] + 76.442;
   1:L PR[91] R[100]mm/sec CNT100;
   1:  PR[91,1] = PR[90,1] + 53.638;
   1:  PR[91,2] = PR[90,2] + 22.256;
   1:  PR[91,3] = PR[90,3] + 76.452;
   1:L PR[91] R[100]mm/sec CNT100;
   1:  PR[91,1] = PR[90,1] + 51.453;
   1:  PR[91,2] = PR[90,2] + 23.180;
   1:  PR[91,3] = PR[90,3] + 76.460;
   1:L PR[91] R[100]mm/sec CNT100;
   1:  PR[91,1] = PR[90,1] + 49.432;
   1:  PR[91,2] = PR[90,2] + 23.965;
   1:  PR[91,3] = PR[90,3] + 76.469;
   1:L PR[91] R[100]mm/sec CNT100;
   1:  PR[91,1] = PR[90,1] + 47.079;
   1:  PR[91,2] = PR[90,2] + 24.601;
   1:  PR[91,3] = PR[90,3] + 76.477;
   1:L PR[91] R[100]mm/sec CNT100;
   1:  PR[91,1] = PR[90,1] + 44.903;
   1:  PR[91,2] = PR[90,2] + 25.331;
   1:  PR[91,3] = PR[90,3] + 76.486;
   1:L PR[91] R[100]mm/sec CNT100;
   1:  PR[91,1] = PR[90,1] + 43.395;
   1:  PR[91,2] = PR[90,2] + 25.692;
   1:  PR[91,3] = PR[90,3] + 76.495;
   1:L PR[91] R[100]mm/sec CNT100;
   1:  PR[91,1] = PR[90,1] + 40.601;
   1:  PR[91,2] = PR[90,2] + 26.173;
   1:  PR[91,3] = PR[90,3] + 76.501;
   1:L PR[91] R[100]mm/sec CNT100;
   1:  PR[91,1] = PR[90,1] + 36.008;
   1:  PR[91,2] = PR[90,2] + 26.528;
   1:  PR[91,3] = PR[90,3] + 76.512;
   1:L PR[91] R[100]mm/sec CNT100;
   1:  PR[91,1] = PR[90,1] + 35.732;
   1:  PR[91,2] = PR[90,2] + 26.532;
   1:  PR[91,3] = PR[90,3] + 76.530;
   1:L PR[91] R[100]mm/sec CNT100;
   1:  PR[91,1] = PR[90,1] + 30.544;
   1:  PR[91,2] = PR[90,2] + 26.116;
   1:  PR[91,3] = PR[90,3] + 76.531;
   1:L PR[91] R[100]mm/sec CNT100;
   1:  PR[91,1] = PR[90,1] + 28.911;
   1:  PR[91,2] = PR[90,2] + 25.742;
   1:  PR[91,3] = PR[90,3] + 76.551;
   1:L PR[91] R[100]mm/sec CNT100;
   1:  PR[91,1] = PR[90,1] + 25.230;
   1:  PR[91,2] = PR[90,2] + 24.781;
   1:  PR[91,3] = PR[90,3] + 76.557;
   1:L PR[91] R[100]mm/sec CNT100;
   1:  PR[91,1] = PR[90,1] + 23.121;
   1:  PR[91,2] = PR[90,2] + 25.099;
   1:  PR[91,3] = PR[90,3] + 76.572;
   1:L PR[91] R[100]mm/sec CNT100;
   1:  PR[91,1] = PR[90,1] + 18.179;
   1:  PR[91,2] = PR[90,2] + 25.258;
   1:  PR[91,3] = PR[90,3] + 76.580;
   1:L PR[91] R[100]mm/sec CNT100;
   1:  PR[91,1] = PR[90,1] + 16.870;
   1:  PR[91,2] = PR[90,2] + 25.205;
   1:  PR[91,3] = PR[90,3] + 76.599;
   1:L PR[91] R[100]mm/sec CNT100;
   1:  PR[91,1] = PR[90,1] + 11.562;
   1:  PR[91,2] = PR[90,2] + 24.060;
   1:  PR[91,3] = PR[90,3] + 76.604;
   1:L PR[91] R[100]mm/sec CNT100;
   1:  PR[91,1] = PR[90,1] + 10.668;
   1:  PR[91,2] = PR[90,2] + 23.817;
   1:  PR[91,3] = PR[90,3] + 76.625;
   1:L PR[91] R[100]mm/sec CNT100;
   1:  PR[91,1] = PR[90,1] + 9.232;
   1:  PR[91,2] = PR[90,2] + 23.158;
   1:  PR[91,3] = PR[90,3] + 76.628;
   1:L PR[91] R[100]mm/sec CNT100;
   1:  PR[91,1] = PR[90,1] + 6.658;
   1:  PR[91,2] = PR[90,2] + 23.820;
   1:  PR[91,3] = PR[90,3] + 76.634;
   1:L PR[91] R[100]mm/sec CNT100;
   1:  PR[91,1] = PR[90,1] + 6.292;
   1:  PR[91,2] = PR[90,2] + 23.894;
   1:  PR[91,3] = PR[90,3] + 76.644;
   1:L PR[91] R[100]mm/sec CNT100;
   1:  PR[91,1] = PR[90,1] + 4.125;
   1:  PR[91,2] = PR[90,2] + 24.151;
   1:  PR[91,3] = PR[90,3] + 76.646;
   1:L PR[91] R[100]mm/sec CNT100;
   1:  PR[91,1] = PR[90,1] + -0.919;
   1:  PR[91,2] = PR[90,2] + 24.504;
   1:  PR[91,3] = PR[90,3] + 76.654;
   1:L PR[91] R[100]mm/sec CNT100;
   1:  PR[91,1] = PR[90,1] + -1.502;
   1:  PR[91,2] = PR[90,2] + 24.503;
   1:  PR[91,3] = PR[90,3] + 76.674;
   1:L PR[91] R[100]mm/sec CNT100;
   1:  PR[91,1] = PR[90,1] + -7.921;
   1:  PR[91,2] = PR[90,2] + 23.871;
   1:  PR[91,3] = PR[90,3] + 76.676;
   1:L PR[91] R[100]mm/sec CNT100;
   1:  PR[91,1] = PR[90,1] + -9.601;
   1:  PR[91,2] = PR[90,2] + 23.477;
   1:  PR[91,3] = PR[90,3] + 76.701;
   1:L PR[91] R[100]mm/sec CNT100;
   1:  PR[91,1] = PR[90,1] + -10.909;
   1:  PR[91,2] = PR[90,2] + 23.656;
   1:  PR[91,3] = PR[90,3] + 76.707;
   1:L PR[91] R[100]mm/sec CNT100;
   1:  PR[91,1] = PR[90,1] + -13.256;
   1:  PR[91,2] = PR[90,2] + 23.913;
   1:  PR[91,3] = PR[90,3] + 76.712;
   1:L PR[91] R[100]mm/sec CNT100;
   1:  PR[91,1] = PR[90,1] + -16.734;
   1:  PR[91,2] = PR[90,2] + 24.232;
   1:  PR[91,3] = PR[90,3] + 76.721;
   1:L PR[91] R[100]mm/sec CNT100;
   1:  PR[91,1] = PR[90,1] + -26.619;
   1:  PR[91,2] = PR[90,2] + 24.602;
   1:  PR[91,3] = PR[90,3] + 76.735;
   1:L PR[91] R[100]mm/sec CNT100;
   1:  PR[91,1] = PR[90,1] + -32.992;
   1:  PR[91,2] = PR[90,2] + 24.411;
   1:  PR[91,3] = PR[90,3] + 76.773;
   1:L PR[91] R[100]mm/sec CNT100;
   1:  PR[91,1] = PR[90,1] + -38.952;
   1:  PR[91,2] = PR[90,2] + 23.902;
   1:  PR[91,3] = PR[90,3] + 76.797;
   1:L PR[91] R[100]mm/sec CNT100;
   1:  PR[91,1] = PR[90,1] + -40.166;
   1:  PR[91,2] = PR[90,2] + 23.822;
   1:  PR[91,3] = PR[90,3] + 76.820;
   1:L PR[91] R[100]mm/sec CNT100;
   1:  PR[91,1] = PR[90,1] + -42.567;
   1:  PR[91,2] = PR[90,2] + 23.411;
   1:  PR[91,3] = PR[90,3] + 76.825;
   1:L PR[91] R[100]mm/sec CNT100;
   1:  PR[91,1] = PR[90,1] + -47.291;
   1:  PR[91,2] = PR[90,2] + 22.501;
   1:  PR[91,3] = PR[90,3] + 76.834;
   1:L PR[91] R[100]mm/sec CNT100;
   1:  PR[91,1] = PR[90,1] + -50.078;
   1:  PR[91,2] = PR[90,2] + 21.634;
   1:  PR[91,3] = PR[90,3] + 76.852;
   1:L PR[91] R[100]mm/sec CNT100;
   1:  PR[91,1] = PR[90,1] + -53.115;
   1:  PR[91,2] = PR[90,2] + 20.640;
   1:  PR[91,3] = PR[90,3] + 76.864;
   1:L PR[91] R[100]mm/sec CNT100;
   1:  PR[91,1] = PR[90,1] + -54.843;
   1:  PR[91,2] = PR[90,2] + 20.012;
   1:  PR[91,3] = PR[90,3] + 76.876;
   1:L PR[91] R[100]mm/sec CNT100;
   1:  PR[91,1] = PR[90,1] + -57.622;
   1:  PR[91,2] = PR[90,2] + 18.557;
   1:  PR[91,3] = PR[90,3] + 76.883;
   1:L PR[91] R[100]mm/sec CNT100;
   1:  PR[91] = PR[90];
   1:  PR[91,1] = PR[90,1] + -59.923;
   1:  PR[91,2] = PR[90,2] + 16.713;
   1:  PR[91,3] = PR[90,3] + 78.195;
   1:L PR[91] R[100]mm/sec CNT100;
   1:  PR[91,1] = PR[90,1] + -61.088;
   1:  PR[91,2] = PR[90,2] + 15.792;
   1:  PR[91,3] = PR[90,3] + 76.908;
   1:L PR[91] R[100]mm/sec CNT100;
   1:  PR[91,1] = PR[90,1] + -64.563;
   1:  PR[91,2] = PR[90,2] + 12.906;
   1:  PR[91,3] = PR[90,3] + 76.914;
   1:L PR[91] R[100]mm/sec CNT100;
   1:  PR[91,1] = PR[90,1] + -64.751;
   1:  PR[91,2] = PR[90,2] + 12.734;
   1:  PR[91,3] = PR[90,3] + 76.931;
   1:L PR[91] R[100]mm/sec CNT100;
   1:  PR[91,1] = PR[90,1] + -67.821;
   1:  PR[91,2] = PR[90,2] + 8.435;
   1:  PR[91,3] = PR[90,3] + 76.932;
   1:L PR[91] R[100]mm/sec CNT100;
   1:  PR[91,1] = PR[90,1] + -69.130;
   1:  PR[91,2] = PR[90,2] + 5.200;
   1:  PR[91,3] = PR[90,3] + 76.953;
   1:L PR[91] R[100]mm/sec CNT100;
   1:  PR[91,1] = PR[90,1] + -69.650;
   1:  PR[91,2] = PR[90,2] + 3.906;
   1:  PR[91,3] = PR[90,3] + 76.966;
   1:L PR[91] R[100]mm/sec CNT100;
   1:  PR[91,1] = PR[90,1] + -69.862;
   1:  PR[91,2] = PR[90,2] + 2.292;
   1:  PR[91,3] = PR[90,3] + 76.972;
   1:L PR[91] R[100]mm/sec CNT100;
   1:  PR[91,1] = PR[90,1] + -70.389;
   1:  PR[91,2] = PR[90,2] + -0.698;
   1:  PR[91,3] = PR[90,3] + 76.978;
   1:L PR[91] R[100]mm/sec CNT100;
   1:  PR[91,1] = PR[90,1] + -70.382;
   1:  PR[91,2] = PR[90,2] + -0.732;
   1:  PR[91,3] = PR[90,3] + 76.990;
   1:L PR[91] R[100]mm/sec CNT100;
   1:  PR[91,1] = PR[90,1] + -69.769;
   1:  PR[91,2] = PR[90,2] + -5.495;
   1:L PR[91] R[100]mm/sec CNT100;
   1:  PR[91,1] = PR[90,1] + -69.452;
   1:  PR[91,2] = PR[90,2] + -6.286;
   1:  PR[91,3] = PR[90,3] + 77.008;
   1:L PR[91] R[100]mm/sec CNT100;
   1:  PR[91,1] = PR[90,1] + -67.800;
   1:  PR[91,2] = PR[90,2] + -10.028;
   1:  PR[91,3] = PR[90,3] + 77.012;
   1:L PR[91] R[100]mm/sec CNT100;
   1:  PR[91,1] = PR[90,1] + -67.559;
   1:  PR[91,2] = PR[90,2] + -10.359;
   1:  PR[91,3] = PR[90,3] + 77.028;
   1:L PR[91] R[100]mm/sec CNT100;
   1:  PR[91,1] = PR[90,1] + -64.570;
   1:  PR[91,2] = PR[90,2] + -14.196;
   1:  PR[91,3] = PR[90,3] + 77.029;
   1:L PR[91] R[100]mm/sec CNT100;
   1:  PR[91,1] = PR[90,1] + -63.011;
   1:  PR[91,2] = PR[90,2] + -15.601;
   1:  PR[91,3] = PR[90,3] + 77.048;
   1:L PR[91] R[100]mm/sec CNT100;
   1:  PR[91,1] = PR[90,1] + -60.356;
   1:  PR[91,2] = PR[90,2] + -17.814;
   1:  PR[91,3] = PR[90,3] + 77.056;
   1:L PR[91] R[100]mm/sec CNT100;
   1:  PR[91,1] = PR[90,1] + -56.217;
   1:  PR[91,2] = PR[90,2] + -20.352;
   1:  PR[91,3] = PR[90,3] + 77.070;
   1:L PR[91] R[100]mm/sec CNT100;
   1:  PR[91,1] = PR[90,1] + -55.448;
   1:  PR[91,2] = PR[90,2] + -20.781;
   1:  PR[91,3] = PR[90,3] + 77.088;
   1:L PR[91] R[100]mm/sec CNT100;
   1:  PR[91,1] = PR[90,1] + -53.919;
   1:  PR[91,2] = PR[90,2] + -21.404;
   1:  PR[91,3] = PR[90,3] + 77.092;
   1:L PR[91] R[100]mm/sec CNT100;
   1:  PR[91,1] = PR[90,1] + -50.274;
   1:  PR[91,2] = PR[90,2] + -22.767;
   1:  PR[91,3] = PR[90,3] + 77.098;
   1:L PR[91] R[100]mm/sec CNT100;
   1:  PR[91,1] = PR[90,1] + -48.085;
   1:  PR[91,2] = PR[90,2] + -23.514;
   1:  PR[91,3] = PR[90,3] + 77.113;
   1:L PR[91] R[100]mm/sec CNT100;
   1:  PR[91,1] = PR[90,1] + -45.017;
   1:  PR[91,2] = PR[90,2] + -24.221;
   1:  PR[91,3] = PR[90,3] + 77.122;
   1:L PR[91] R[100]mm/sec CNT100;
   1:  PR[91,1] = PR[90,1] + -40.786;
   1:  PR[91,2] = PR[90,2] + -25.052;
   1:  PR[91,3] = PR[90,3] + 77.134;
   1:L PR[91] R[100]mm/sec CNT100;
   1:  PR[91,1] = PR[90,1] + -38.694;
   1:  PR[91,2] = PR[90,2] + -25.441;
   1:  PR[91,3] = PR[90,3] + 77.151;
   1:L PR[91] R[100]mm/sec CNT100;
   1:  PR[91,1] = PR[90,1] + -36.027;
   1:  PR[91,2] = PR[90,2] + -25.726;
   1:  PR[91,3] = PR[90,3] + 77.159;
   1:L PR[91] R[100]mm/sec CNT100;
   1:  PR[91,1] = PR[90,1] + -31.850;
   1:  PR[91,2] = PR[90,2] + -26.059;
   1:  PR[91,3] = PR[90,3] + 77.170;
   1:L PR[91] R[100]mm/sec CNT100;
   1:  PR[91,1] = PR[90,1] + -23.988;
   1:  PR[91,2] = PR[90,2] + -26.313;
   1:  PR[91,3] = PR[90,3] + 77.186;
   1:L PR[91] R[100]mm/sec CNT100;
   1:  PR[91,1] = PR[90,1] + -14.147;
   1:  PR[91,2] = PR[90,2] + -25.955;
   1:  PR[91,3] = PR[90,3] + 77.217;
   1:L PR[91] R[100]mm/sec CNT100;
   1:  PR[91,1] = PR[90,1] + -13.688;
   1:  PR[91,2] = PR[90,2] + -25.922;
   1:  PR[91,3] = PR[90,3] + 77.255;
   1:L PR[91] R[100]mm/sec CNT100;
   1:  PR[91,1] = PR[90,1] + -9.685;
   1:  PR[91,2] = PR[90,2] + -25.467;
   1:  PR[91,3] = PR[90,3] + 77.257;
   1:L PR[91] R[100]mm/sec CNT100;
   1:  PR[91,1] = PR[90,1] + -8.709;
   1:  PR[91,2] = PR[90,2] + -25.441;
   1:  PR[91,3] = PR[90,3] + 77.272;
   1:L PR[91] R[100]mm/sec CNT100;
   1:  PR[91,1] = PR[90,1] + -7.981;
   1:  PR[91,2] = PR[90,2] + -25.351;
   1:  PR[91,3] = PR[90,3] + 77.276;
   1:L PR[91] R[100]mm/sec CNT100;
   1:  PR[91,1] = PR[90,1] + -7.226;
   1:  PR[91,2] = PR[90,2] + -25.528;
   1:  PR[91,3] = PR[90,3] + 77.279;
   1:L PR[91] R[100]mm/sec CNT100;
   1:  PR[91,1] = PR[90,1] + -5.779;
   1:  PR[91,2] = PR[90,2] + -25.667;
   1:  PR[91,3] = PR[90,3] + 77.282;
   1:L PR[91] R[100]mm/sec CNT100;
   1:  PR[91,1] = PR[90,1] + -1.148;
   1:  PR[91,2] = PR[90,2] + -26.158;
   1:  PR[91,3] = PR[90,3] + 77.287;
   1:L PR[91] R[100]mm/sec CNT100;
   1:  PR[91,1] = PR[90,1] + -0.859;
   1:  PR[91,2] = PR[90,2] + -26.177;
   1:  PR[91,3] = PR[90,3] + 77.306;
   1:L PR[91] R[100]mm/sec CNT100;
   1:  PR[91,1] = PR[90,1] + 0.581;
   1:  PR[91,2] = PR[90,2] + -26.180;
   1:  PR[91,3] = PR[90,3] + 77.307;
   1:L PR[91] R[100]mm/sec CNT100;
   1:  PR[91,1] = PR[90,1] + 4.613;
   1:  PR[91,2] = PR[90,2] + -25.901;
   1:  PR[91,3] = PR[90,3] + 77.312;
   1:L PR[91] R[100]mm/sec CNT100;
   1:  PR[91,1] = PR[90,1] + 7.461;
   1:  PR[91,2] = PR[90,2] + -25.564;
   1:  PR[91,3] = PR[90,3] + 77.328;
   1:L PR[91] R[100]mm/sec CNT100;
   1:  PR[91,1] = PR[90,1] + 7.983;
   1:  PR[91,2] = PR[90,2] + -25.458;
   1:  PR[91,3] = PR[90,3] + 77.339;
   1:L PR[91] R[100]mm/sec CNT100;
   1:  PR[91,1] = PR[90,1] + 9.579;
   1:  PR[91,2] = PR[90,2] + -25.048;
   1:  PR[91,3] = PR[90,3] + 77.341;
   1:L PR[91] R[100]mm/sec CNT100;
   1:  PR[91,1] = PR[90,1] + 10.535;
   1:  PR[91,2] = PR[90,2] + -25.487;
   1:  PR[91,3] = PR[90,3] + 77.347;
   1:L PR[91] R[100]mm/sec CNT100;
   1:  PR[91,1] = PR[90,1] + 10.865;
   1:  PR[91,2] = PR[90,2] + -25.577;
   1:  PR[91,3] = PR[90,3] + 77.352;
   1:L PR[91] R[100]mm/sec CNT100;
   1:  PR[91,1] = PR[90,1] + 16.833;
   1:  PR[91,2] = PR[90,2] + -26.865;
   1:  PR[91,3] = PR[90,3] + 77.353;
   1:L PR[91] R[100]mm/sec CNT100;
   1:  PR[91,1] = PR[90,1] + 17.573;
   1:  PR[91,2] = PR[90,2] + -26.895;
   1:  PR[91,3] = PR[90,3] + 77.377;
   1:L PR[91] R[100]mm/sec CNT100;
   1:  PR[91,1] = PR[90,1] + 23.172;
   1:  PR[91,2] = PR[90,2] + -26.714;
   1:  PR[91,3] = PR[90,3] + 77.379;
   1:L PR[91] R[100]mm/sec CNT100;
   1:  PR[91,1] = PR[90,1] + 24.763;
   1:  PR[91,2] = PR[90,2] + -26.476;
   1:  PR[91,3] = PR[90,3] + 77.401;
   1:L PR[91] R[100]mm/sec CNT100;
   1:  PR[91,1] = PR[90,1] + 27.460;
   1:  PR[91,2] = PR[90,2] + -27.180;
   1:  PR[91,3] = PR[90,3] + 77.407;
   1:L PR[91] R[100]mm/sec CNT100;
   1:  PR[91,1] = PR[90,1] + 30.172;
   1:  PR[91,2] = PR[90,2] + -27.801;
   1:  PR[91,3] = PR[90,3] + 77.418;
   1:L PR[91] R[100]mm/sec CNT100;
   1:  PR[91,1] = PR[90,1] + 34.661;
   1:  PR[91,2] = PR[90,2] + -28.160;
   1:  PR[91,3] = PR[90,3] + 77.429;
   1:L PR[91] R[100]mm/sec CNT100;
   1:  PR[91,1] = PR[90,1] + 35.284;
   1:  PR[91,2] = PR[90,2] + -28.195;
   1:  PR[91,3] = PR[90,3] + 77.446;
   1:L PR[91] R[100]mm/sec CNT100;
   1:  PR[91,1] = PR[90,1] + 36.831;
   1:  PR[91,2] = PR[90,2] + -28.047;
   1:  PR[91,3] = PR[90,3] + 77.449;
   1:L PR[91] R[100]mm/sec CNT100;
   1:  PR[91,1] = PR[90,1] + 40.358;
   1:  PR[91,2] = PR[90,2] + -27.775;
   1:  PR[91,3] = PR[90,3] + 77.455;
   1:L PR[91] R[100]mm/sec CNT100;
   1:  PR[91,1] = PR[90,1] + 41.931;
   1:  PR[91,2] = PR[90,2] + -27.504;
   1:  PR[91,3] = PR[90,3] + 77.469;
   1:L PR[91] R[100]mm/sec CNT100;
   1:  PR[91,1] = PR[90,1] + 44.773;
   1:  PR[91,2] = PR[90,2] + -26.824;
   1:  PR[91,3] = PR[90,3] + 77.475;
   1:L PR[91] R[100]mm/sec CNT100;
   1:  PR[91,1] = PR[90,1] + 48.715;
   1:  PR[91,2] = PR[90,2] + -25.508;
   1:  PR[91,3] = PR[90,3] + 77.486;
   1:L PR[91] R[100]mm/sec CNT100;
   1:  PR[91,1] = PR[90,1] + 53.139;
   1:  PR[91,2] = PR[90,2] + -23.641;
   1:  PR[91,3] = PR[90,3] + 77.502;
   1:L PR[91] R[100]mm/sec CNT100;
   1:  PR[91,1] = PR[90,1] + 56.598;
   1:  PR[91,2] = PR[90,2] + -21.735;
   1:  PR[91,3] = PR[90,3] + 77.521;
   1:L PR[91] R[100]mm/sec CNT100;
   1:  PR[91,1] = PR[90,1] + 56.791;
   1:  PR[91,2] = PR[90,2] + -21.644;
   1:  PR[91,3] = PR[90,3] + 77.536;
   1:L PR[91] R[100]mm/sec CNT100;
   1:  PR[91,1] = PR[90,1] + 60.697;
   1:  PR[91,2] = PR[90,2] + -19.149;
   1:  PR[91,3] = PR[90,3] + 77.537;
   1:L PR[91] R[100]mm/sec CNT100;
   1:  PR[91,1] = PR[90,1] + 62.864;
   1:  PR[91,2] = PR[90,2] + -17.319;
   1:  PR[91,3] = PR[90,3] + 77.555;
   1:L PR[91] R[100]mm/sec CNT100;
   1:  PR[91,1] = PR[90,1] + 64.236;
   1:  PR[91,2] = PR[90,2] + -16.111;
   1:  PR[91,3] = PR[90,3] + 77.566;
   1:L PR[91] R[100]mm/sec CNT100;
   1:  PR[91,1] = PR[90,1] + 67.448;
   1:  PR[91,2] = PR[90,2] + -12.111;
   1:  PR[91,3] = PR[90,3] + 77.573;
   1:L PR[91] R[100]mm/sec CNT100;
   1:  PR[91,1] = PR[90,1] + 68.762;
   1:  PR[91,2] = PR[90,2] + -9.747;
   1:  PR[91,3] = PR[90,3] + 77.593;
   1:L PR[91] R[100]mm/sec CNT100;
   1:  PR[91,1] = PR[90,1] + 69.760;
   1:  PR[91,2] = PR[90,2] + -7.466;
   1:  PR[91,3] = PR[90,3] + 77.603;
   1:L PR[91] R[100]mm/sec CNT100;
   1:  PR[91,1] = PR[90,1] + 70.405;
   1:  PR[91,2] = PR[90,2] + -5.465;
   1:  PR[91,3] = PR[90,3] + 77.613;
   1:L PR[91] R[100]mm/sec CNT100;
   1:  PR[91,1] = PR[90,1] + 70.823;
   1:  PR[91,2] = PR[90,2] + -2.539;
   1:  PR[91,3] = PR[90,3] + 77.621;
   1:L PR[91] R[100]mm/sec CNT100;
   1:  PR[91,1] = PR[90,1] + 71.010;
   1:  PR[91,2] = PR[90,2] + -0.768;
   1:  PR[91,3] = PR[90,3] + 77.633;
   1:L PR[91] R[100]mm/sec CNT100;
   1:  PR[91,1] = PR[90,1] + 70.594;
   1:  PR[91,2] = PR[90,2] + 2.114;
   1:  PR[91,3] = PR[90,3] + 77.640;
   1:L PR[91] R[100]mm/sec CNT100;
   1:  PR[91,1] = PR[90,1] + 70.394;
   1:  PR[91,2] = PR[90,2] + 4.041;
   1:  PR[91,3] = PR[90,3] + 77.651;
   1:L PR[91] R[100]mm/sec CNT100;
   1:  PR[91,1] = PR[90,1] + 69.761;
   1:  PR[91,2] = PR[90,2] + 6.006;
   1:  PR[91,3] = PR[90,3] + 77.658;
   1:L PR[91] R[100]mm/sec CNT100;
   1:  PR[91,1] = PR[90,1] + 68.763;
   1:  PR[91,2] = PR[90,2] + 8.286;
   1:  PR[91,3] = PR[90,3] + 77.666;
   1:L PR[91] R[100]mm/sec CNT100;
   1:  PR[91,1] = PR[90,1] + 67.443;
   1:  PR[91,2] = PR[90,2] + 10.661;
   1:  PR[91,3] = PR[90,3] + 77.676;
   1:L PR[91] R[100]mm/sec CNT100;
   1:  PR[91,1] = PR[90,1] + 66.473;
   1:  PR[91,2] = PR[90,2] + 11.902;
   1:  PR[91,3] = PR[90,3] + 77.687;
   1:L PR[91] R[100]mm/sec CNT100;
   1:  PR[91,1] = PR[90,1] + 64.242;
   1:  PR[91,2] = PR[90,2] + 14.647;
   1:  PR[91,3] = PR[90,3] + 77.693;
   1:L PR[91] R[100]mm/sec CNT100;
   1:  PR[91,1] = PR[90,1] + 62.864;
   1:  PR[91,2] = PR[90,2] + 15.860;
   1:  PR[91,3] = PR[90,3] + 77.706;
   1:L PR[91] R[100]mm/sec CNT100;
   1:  PR[91,1] = PR[90,1] + 60.697;
   1:  PR[91,2] = PR[90,2] + 17.690;
   1:  PR[91,3] = PR[90,3] + 77.714;
   1:L PR[91] R[100]mm/sec CNT100;
   1:  PR[91,1] = PR[90,1] + 56.791;
   1:  PR[91,2] = PR[90,2] + 20.186;
   1:  PR[91,3] = PR[90,3] + 77.725;
   1:L PR[91] R[100]mm/sec CNT100;
   1:  PR[91,1] = PR[90,1] + 56.598;
   1:  PR[91,2] = PR[90,2] + 20.276;
   1:  PR[91,3] = PR[90,3] + 77.743;
   1:L PR[91] R[100]mm/sec CNT100;
   1:  PR[91,1] = PR[90,1] + 53.139;
   1:  PR[91,2] = PR[90,2] + 22.182;
   1:L PR[91] R[100]mm/sec CNT100;
   1:  PR[91,1] = PR[90,1] + 48.715;
   1:  PR[91,2] = PR[90,2] + 24.049;
   1:  PR[91,3] = PR[90,3] + 77.759;
   1:L PR[91] R[100]mm/sec CNT100;
   1:  PR[91,1] = PR[90,1] + 44.774;
   1:  PR[91,2] = PR[90,2] + 25.365;
   1:  PR[91,3] = PR[90,3] + 77.777;
   1:L PR[91] R[100]mm/sec CNT100;
   1:  PR[91,1] = PR[90,1] + 41.931;
   1:  PR[91,2] = PR[90,2] + 26.046;
   1:  PR[91,3] = PR[90,3] + 77.793;
   1:L PR[91] R[100]mm/sec CNT100;
   1:  PR[91,1] = PR[90,1] + 40.358;
   1:  PR[91,2] = PR[90,2] + 26.316;
   1:  PR[91,3] = PR[90,3] + 77.805;
   1:L PR[91] R[100]mm/sec CNT100;
   1:  PR[91,1] = PR[90,1] + 36.831;
   1:  PR[91,2] = PR[90,2] + 26.588;
   1:  PR[91,3] = PR[90,3] + 77.811;
   1:L PR[91] R[100]mm/sec CNT100;
   1:  PR[91,1] = PR[90,1] + 35.284;
   1:  PR[91,2] = PR[90,2] + 26.737;
   1:  PR[91,3] = PR[90,3] + 77.825;
   1:L PR[91] R[100]mm/sec CNT100;
   1:  PR[91,1] = PR[90,1] + 34.661;
   1:  PR[91,2] = PR[90,2] + 26.702;
   1:  PR[91,3] = PR[90,3] + 77.831;
   1:L PR[91] R[100]mm/sec CNT100;
   1:  PR[91,1] = PR[90,1] + 30.172;
   1:  PR[91,2] = PR[90,2] + 26.343;
   1:  PR[91,3] = PR[90,3] + 77.833;
   1:L PR[91] R[100]mm/sec CNT100;
   1:  PR[91,1] = PR[90,1] + 27.461;
   1:  PR[91,2] = PR[90,2] + 25.721;
   1:  PR[91,3] = PR[90,3] + 77.851;
   1:L PR[91] R[100]mm/sec CNT100;
   1:  PR[91,1] = PR[90,1] + 24.763;
   1:  PR[91,2] = PR[90,2] + 25.017;
   1:  PR[91,3] = PR[90,3] + 77.861;
   1:L PR[91] R[100]mm/sec CNT100;
   1:  PR[91,1] = PR[90,1] + 23.172;
   1:  PR[91,2] = PR[90,2] + 25.256;
   1:  PR[91,3] = PR[90,3] + 77.872;
   1:L PR[91] R[100]mm/sec CNT100;
   1:  PR[91,1] = PR[90,1] + 17.573;
   1:  PR[91,2] = PR[90,2] + 25.436;
   1:  PR[91,3] = PR[90,3] + 77.878;
   1:L PR[91] R[100]mm/sec CNT100;
   1:  PR[91,1] = PR[90,1] + 16.833;
   1:  PR[91,2] = PR[90,2] + 25.406;
   1:  PR[91,3] = PR[90,3] + 77.900;
   1:L PR[91] R[100]mm/sec CNT100;
   1:  PR[91,1] = PR[90,1] + 10.865;
   1:  PR[91,2] = PR[90,2] + 24.118;
   1:  PR[91,3] = PR[90,3] + 77.903;
   1:L PR[91] R[100]mm/sec CNT100;
   1:  PR[91,1] = PR[90,1] + 10.534;
   1:  PR[91,2] = PR[90,2] + 24.028;
   1:  PR[91,3] = PR[90,3] + 77.927;
   1:L PR[91] R[100]mm/sec CNT100;
   1:  PR[91,1] = PR[90,1] + 9.578;
   1:  PR[91,2] = PR[90,2] + 23.589;
   1:  PR[91,3] = PR[90,3] + 77.928;
   1:L PR[91] R[100]mm/sec CNT100;
   1:  PR[91,1] = PR[90,1] + 7.992;
   1:  PR[91,2] = PR[90,2] + 23.998;
   1:  PR[91,3] = PR[90,3] + 77.932;
   1:L PR[91] R[100]mm/sec CNT100;
   1:  PR[91,1] = PR[90,1] + 7.478;
   1:  PR[91,2] = PR[90,2] + 24.102;
   1:  PR[91,3] = PR[90,3] + 77.938;
   1:L PR[91] R[100]mm/sec CNT100;
   1:  PR[91,1] = PR[90,1] + 4.632;
   1:  PR[91,2] = PR[90,2] + 24.439;
   1:  PR[91,3] = PR[90,3] + 77.940;
   1:L PR[91] R[100]mm/sec CNT100;
   1:  PR[91,1] = PR[90,1] + 0.604;
   1:  PR[91,2] = PR[90,2] + 24.721;
   1:  PR[91,3] = PR[90,3] + 77.952;
   1:L PR[91] R[100]mm/sec CNT100;
   1:  PR[91,1] = PR[90,1] + -0.800;
   1:  PR[91,2] = PR[90,2] + 24.718;
   1:  PR[91,3] = PR[90,3] + 77.967;
   1:L PR[91] R[100]mm/sec CNT100;
   1:  PR[91,1] = PR[90,1] + -7.222;
   1:  PR[91,2] = PR[90,2] + 24.070;
   1:  PR[91,3] = PR[90,3] + 77.973;
   1:L PR[91] R[100]mm/sec CNT100;
   1:  PR[91,1] = PR[90,1] + -7.972;
   1:  PR[91,2] = PR[90,2] + 23.894;
   1:  PR[91,3] = PR[90,3] + 77.998;
   1:L PR[91] R[100]mm/sec CNT100;
   1:  PR[91,1] = PR[90,1] + -9.821;
   1:  PR[91,2] = PR[90,2] + 24.106;
   1:  PR[91,3] = PR[90,3] + 78.001;
   1:L PR[91] R[100]mm/sec CNT100;
   1:  PR[91,1] = PR[90,1] + -13.981;
   1:  PR[91,2] = PR[90,2] + 24.484;
   1:  PR[91,3] = PR[90,3] + 78.008;
   1:L PR[91] R[100]mm/sec CNT100;
   1:  PR[91,1] = PR[90,1] + -23.990;
   1:  PR[91,2] = PR[90,2] + 24.854;
   1:  PR[91,3] = PR[90,3] + 78.024;
   1:L PR[91] R[100]mm/sec CNT100;
   1:  PR[91,1] = PR[90,1] + -31.838;
   1:  PR[91,2] = PR[90,2] + 24.605;
   1:  PR[91,3] = PR[90,3] + 78.063;
   1:L PR[91] R[100]mm/sec CNT100;
   1:  PR[91,1] = PR[90,1] + -37.491;
   1:  PR[91,2] = PR[90,2] + 24.122;
   1:  PR[91,3] = PR[90,3] + 78.093;
   1:L PR[91] R[100]mm/sec CNT100;
   1:  PR[91,1] = PR[90,1] + -38.823;
   1:  PR[91,2] = PR[90,2] + 23.982;
   1:  PR[91,3] = PR[90,3] + 78.115;
   1:L PR[91] R[100]mm/sec CNT100;
   1:  PR[91,1] = PR[90,1] + -46.088;
   1:  PR[91,2] = PR[90,2] + 22.585;
   1:  PR[91,3] = PR[90,3] + 78.121;
   1:L PR[91] R[100]mm/sec CNT100;
   1:  PR[91,1] = PR[90,1] + -51.135;
   1:  PR[91,2] = PR[90,2] + 21.016;
   1:  PR[91,3] = PR[90,3] + 78.149;
   1:L PR[91] R[100]mm/sec CNT100;
   1:  PR[91,1] = PR[90,1] + -52.570;
   1:  PR[91,2] = PR[90,2] + 20.546;
   1:  PR[91,3] = PR[90,3] + 78.170;
   1:L PR[91] R[100]mm/sec CNT100;
   1:  PR[91,1] = PR[90,1] + -53.318;
   1:  PR[91,2] = PR[90,2] + 20.274;
   1:  PR[91,3] = PR[90,3] + 78.176;
   1:L PR[91] R[100]mm/sec CNT100;
   1:  PR[91,1] = PR[90,1] + -57.031;
   1:  PR[91,2] = PR[90,2] + 18.331;
   1:  PR[91,3] = PR[90,3] + 78.179;
   1:L PR[91] R[100]mm/sec CNT100;
   1:  PR[91] = PR[90];
   1:  PR[91,1] = PR[90,1] + -58.525;
   1:  PR[91,2] = PR[90,2] + 16.939;
   1:  PR[91,3] = PR[90,3] + 79.495;
   1:L PR[91] R[100]mm/sec CNT100;
   1:  PR[91,1] = PR[90,1] + -60.424;
   1:  PR[91,2] = PR[90,2] + 15.436;
   1:  PR[91,3] = PR[90,3] + 78.204;
   1:L PR[91] R[100]mm/sec CNT100;
   1:  PR[91,1] = PR[90,1] + -63.571;
   1:  PR[91,2] = PR[90,2] + 12.823;
   1:  PR[91,3] = PR[90,3] + 78.214;
   1:L PR[91] R[100]mm/sec CNT100;
   1:  PR[91,1] = PR[90,1] + -63.889;
   1:  PR[91,2] = PR[90,2] + 12.432;
   1:  PR[91,3] = PR[90,3] + 78.230;
   1:L PR[91] R[100]mm/sec CNT100;
   1:  PR[91,1] = PR[90,1] + -65.592;
   1:  PR[91,2] = PR[90,2] + 10.265;
   1:  PR[91,3] = PR[90,3] + 78.232;
   1:L PR[91] R[100]mm/sec CNT100;
   1:  PR[91,1] = PR[90,1] + -66.841;
   1:  PR[91,2] = PR[90,2] + 8.515;
   1:  PR[91,3] = PR[90,3] + 78.243;
   1:L PR[91] R[100]mm/sec CNT100;
   1:  PR[91,1] = PR[90,1] + -68.688;
   1:  PR[91,2] = PR[90,2] + 3.945;
   1:  PR[91,3] = PR[90,3] + 78.251;
   1:L PR[91] R[100]mm/sec CNT100;
   1:  PR[91,1] = PR[90,1] + -68.804;
   1:  PR[91,2] = PR[90,2] + 3.058;
   1:  PR[91,3] = PR[90,3] + 78.271;
   1:L PR[91] R[100]mm/sec CNT100;
   1:  PR[91,1] = PR[90,1] + -69.318;
   1:  PR[91,2] = PR[90,2] + 0.144;
   1:  PR[91,3] = PR[90,3] + 78.274;
   1:L PR[91] R[100]mm/sec CNT100;
   1:  PR[91,1] = PR[90,1] + -69.436;
   1:  PR[91,2] = PR[90,2] + -0.725;
   1:  PR[91,3] = PR[90,3] + 78.286;
   1:L PR[91] R[100]mm/sec CNT100;
   1:  PR[91,1] = PR[90,1] + -68.966;
   1:  PR[91,2] = PR[90,2] + -4.088;
   1:  PR[91,3] = PR[90,3] + 78.289;
   1:L PR[91] R[100]mm/sec CNT100;
   1:  PR[91,1] = PR[90,1] + -68.850;
   1:  PR[91,2] = PR[90,2] + -4.728;
   1:  PR[91,3] = PR[90,3] + 78.302;
   1:L PR[91] R[100]mm/sec CNT100;
   1:  PR[91,1] = PR[90,1] + -68.758;
   1:  PR[91,2] = PR[90,2] + -5.058;
   1:  PR[91,3] = PR[90,3] + 78.305;
   1:L PR[91] R[100]mm/sec CNT100;
   1:  PR[91,1] = PR[90,1] + -68.702;
   1:  PR[91,2] = PR[90,2] + -5.478;
   1:  PR[91,3] = PR[90,3] + 78.306;
   1:L PR[91] R[100]mm/sec CNT100;
   1:  PR[91,1] = PR[90,1] + -68.557;
   1:  PR[91,2] = PR[90,2] + -5.829;
   1:  PR[91,3] = PR[90,3] + 78.308;
   1:L PR[91] R[100]mm/sec CNT100;
   1:  PR[91,1] = PR[90,1] + -66.711;
   1:  PR[91,2] = PR[90,2] + -10.010;
   1:  PR[91,3] = PR[90,3] + 78.309;
   1:L PR[91] R[100]mm/sec CNT100;
   1:  PR[91,1] = PR[90,1] + -65.919;
   1:  PR[91,2] = PR[90,2] + -11.101;
   1:  PR[91,3] = PR[90,3] + 78.327;
   1:L PR[91] R[100]mm/sec CNT100;
   1:  PR[91,1] = PR[90,1] + -63.520;
   1:  PR[91,2] = PR[90,2] + -14.179;
   1:  PR[91,3] = PR[90,3] + 78.333;
   1:L PR[91] R[100]mm/sec CNT100;
   1:  PR[91,1] = PR[90,1] + -61.156;
   1:  PR[91,2] = PR[90,2] + -16.312;
   1:  PR[91,3] = PR[90,3] + 78.348;
   1:L PR[91] R[100]mm/sec CNT100;
   1:  PR[91,1] = PR[90,1] + -59.358;
   1:  PR[91,2] = PR[90,2] + -17.811;
   1:  PR[91,3] = PR[90,3] + 78.360;
   1:L PR[91] R[100]mm/sec CNT100;
   1:  PR[91,1] = PR[90,1] + -54.757;
   1:  PR[91,2] = PR[90,2] + -20.631;
   1:  PR[91,3] = PR[90,3] + 78.370;
   1:L PR[91] R[100]mm/sec CNT100;
   1:  PR[91,1] = PR[90,1] + -54.388;
   1:  PR[91,2] = PR[90,2] + -20.832;
   1:  PR[91,3] = PR[90,3] + 78.391;
   1:L PR[91] R[100]mm/sec CNT100;
   1:  PR[91,1] = PR[90,1] + -49.506;
   1:  PR[91,2] = PR[90,2] + -22.657;
   1:  PR[91,3] = PR[90,3] + 78.393;
   1:L PR[91] R[100]mm/sec CNT100;
   1:  PR[91,1] = PR[90,1] + -46.142;
   1:  PR[91,2] = PR[90,2] + -23.805;
   1:  PR[91,3] = PR[90,3] + 78.413;
   1:L PR[91] R[100]mm/sec CNT100;
   1:  PR[91,1] = PR[90,1] + -44.274;
   1:  PR[91,2] = PR[90,2] + -24.235;
   1:  PR[91,3] = PR[90,3] + 78.427;
   1:L PR[91] R[100]mm/sec CNT100;
   1:  PR[91,1] = PR[90,1] + -41.647;
   1:  PR[91,2] = PR[90,2] + -24.752;
   1:  PR[91,3] = PR[90,3] + 78.434;
   1:L PR[91] R[100]mm/sec CNT100;
   1:  PR[91,1] = PR[90,1] + -37.159;
   1:  PR[91,2] = PR[90,2] + -25.586;
   1:  PR[91,3] = PR[90,3] + 78.445;
   1:L PR[91] R[100]mm/sec CNT100;
   1:  PR[91,1] = PR[90,1] + -31.449;
   1:  PR[91,2] = PR[90,2] + -26.196;
   1:  PR[91,3] = PR[90,3] + 78.463;
   1:L PR[91] R[100]mm/sec CNT100;
   1:  PR[91,1] = PR[90,1] + -30.691;
   1:  PR[91,2] = PR[90,2] + -26.257;
   1:  PR[91,3] = PR[90,3] + 78.485;
   1:L PR[91] R[100]mm/sec CNT100;
   1:  PR[91,1] = PR[90,1] + -21.356;
   1:  PR[91,2] = PR[90,2] + -26.566;
   1:  PR[91,3] = PR[90,3] + 78.488;
   1:L PR[91] R[100]mm/sec CNT100;
   1:  PR[91,1] = PR[90,1] + -18.618;
   1:  PR[91,2] = PR[90,2] + -26.480;
   1:  PR[91,3] = PR[90,3] + 78.525;
   1:L PR[91] R[100]mm/sec CNT100;
   1:  PR[91,1] = PR[90,1] + -11.437;
   1:  PR[91,2] = PR[90,2] + -26.211;
   1:  PR[91,3] = PR[90,3] + 78.536;
   1:L PR[91] R[100]mm/sec CNT100;
   1:  PR[91,1] = PR[90,1] + -10.861;
   1:  PR[91,2] = PR[90,2] + -26.169;
   1:  PR[91,3] = PR[90,3] + 78.564;
   1:L PR[91] R[100]mm/sec CNT100;
   1:  PR[91,1] = PR[90,1] + -7.616;
   1:  PR[91,2] = PR[90,2] + -25.801;
   1:  PR[91,3] = PR[90,3] + 78.566;
   1:L PR[91] R[100]mm/sec CNT100;
   1:  PR[91,1] = PR[90,1] + -6.348;
   1:  PR[91,2] = PR[90,2] + -25.766;
   1:  PR[91,3] = PR[90,3] + 78.579;
   1:L PR[91] R[100]mm/sec CNT100;
   1:  PR[91,1] = PR[90,1] + -0.655;
   1:  PR[91,2] = PR[90,2] + -26.360;
   1:  PR[91,3] = PR[90,3] + 78.584;
   1:L PR[91] R[100]mm/sec CNT100;
   1:  PR[91,1] = PR[90,1] + -0.158;
   1:  PR[91,2] = PR[90,2] + -26.392;
   1:  PR[91,3] = PR[90,3] + 78.607;
   1:L PR[91] R[100]mm/sec CNT100;
   1:  PR[91,1] = PR[90,1] + 2.110;
   1:  PR[91,2] = PR[90,2] + -26.397;
   1:  PR[91,3] = PR[90,3] + 78.608;
   1:L PR[91] R[100]mm/sec CNT100;
   1:  PR[91,1] = PR[90,1] + 5.125;
   1:  PR[91,2] = PR[90,2] + -26.188;
   1:  PR[91,3] = PR[90,3] + 78.617;
   1:L PR[91] R[100]mm/sec CNT100;
   1:  PR[91,1] = PR[90,1] + 8.656;
   1:  PR[91,2] = PR[90,2] + -25.770;
   1:  PR[91,3] = PR[90,3] + 78.629;
   1:L PR[91] R[100]mm/sec CNT100;
   1:  PR[91,1] = PR[90,1] + 9.750;
   1:  PR[91,2] = PR[90,2] + -25.548;
   1:  PR[91,3] = PR[90,3] + 78.643;
   1:L PR[91] R[100]mm/sec CNT100;
   1:  PR[91,1] = PR[90,1] + 16.795;
   1:  PR[91,2] = PR[90,2] + -27.065;
   1:  PR[91,3] = PR[90,3] + 78.648;
   1:L PR[91] R[100]mm/sec CNT100;
   1:  PR[91,1] = PR[90,1] + 16.968;
   1:  PR[91,2] = PR[90,2] + -27.072;
   1:  PR[91,3] = PR[90,3] + 78.676;
   1:L PR[91] R[100]mm/sec CNT100;
   1:  PR[91,1] = PR[90,1] + 23.224;
   1:  PR[91,2] = PR[90,2] + -26.871;
   1:  PR[91,3] = PR[90,3] + 78.677;
   1:L PR[91] R[100]mm/sec CNT100;
   1:  PR[91,1] = PR[90,1] + 24.298;
   1:  PR[91,2] = PR[90,2] + -26.713;
   1:  PR[91,3] = PR[90,3] + 78.701;
   1:L PR[91] R[100]mm/sec CNT100;
   1:  PR[91,1] = PR[90,1] + 26.009;
   1:  PR[91,2] = PR[90,2] + -27.159;
   1:  PR[91,3] = PR[90,3] + 78.705;
   1:L PR[91] R[100]mm/sec CNT100;
   1:  PR[91,1] = PR[90,1] + 29.800;
   1:  PR[91,2] = PR[90,2] + -28.028;
   1:  PR[91,3] = PR[90,3] + 78.712;
   1:L PR[91] R[100]mm/sec CNT100;
   1:  PR[91,1] = PR[90,1] + 33.069;
   1:  PR[91,2] = PR[90,2] + -28.289;
   1:  PR[91,3] = PR[90,3] + 78.728;
   1:L PR[91] R[100]mm/sec CNT100;
   1:  PR[91,1] = PR[90,1] + 34.948;
   1:  PR[91,2] = PR[90,2] + -28.395;
   1:  PR[91,3] = PR[90,3] + 78.740;
   1:L PR[91] R[100]mm/sec CNT100;
   1:  PR[91,1] = PR[90,1] + 39.134;
   1:  PR[91,2] = PR[90,2] + -27.994;
   1:  PR[91,3] = PR[90,3] + 78.748;
   1:L PR[91] R[100]mm/sec CNT100;
   1:  PR[91,1] = PR[90,1] + 40.116;
   1:  PR[91,2] = PR[90,2] + -27.918;
   1:  PR[91,3] = PR[90,3] + 78.764;
   1:L PR[91] R[100]mm/sec CNT100;
   1:  PR[91,1] = PR[90,1] + 40.467;
   1:  PR[91,2] = PR[90,2] + -27.858;
   1:  PR[91,3] = PR[90,3] + 78.768;
   1:L PR[91] R[100]mm/sec CNT100;
   1:  PR[91,1] = PR[90,1] + 44.640;
   1:  PR[91,2] = PR[90,2] + -26.858;
   1:  PR[91,3] = PR[90,3] + 78.770;
   1:L PR[91] R[100]mm/sec CNT100;
   1:  PR[91,1] = PR[90,1] + 47.413;
   1:  PR[91,2] = PR[90,2] + -25.928;
   1:  PR[91,3] = PR[90,3] + 78.786;
   1:L PR[91] R[100]mm/sec CNT100;
   1:  PR[91,1] = PR[90,1] + 48.507;
   1:  PR[91,2] = PR[90,2] + -25.470;
   1:  PR[91,3] = PR[90,3] + 78.798;
   1:L PR[91] R[100]mm/sec CNT100;
   1:  PR[91,1] = PR[90,1] + 50.085;
   1:  PR[91,2] = PR[90,2] + -24.647;
   1:  PR[91,3] = PR[90,3] + 78.803;
   1:L PR[91] R[100]mm/sec CNT100;
   1:  PR[91,1] = PR[90,1] + 52.639;
   1:  PR[91,2] = PR[90,2] + -23.567;
   1:  PR[91,3] = PR[90,3] + 78.810;
   1:L PR[91] R[100]mm/sec CNT100;
   1:  PR[91,1] = PR[90,1] + 54.654;
   1:  PR[91,2] = PR[90,2] + -22.457;
   1:  PR[91,3] = PR[90,3] + 78.820;
   1:L PR[91] R[100]mm/sec CNT100;
   1:  PR[91,1] = PR[90,1] + 56.192;
   1:  PR[91,2] = PR[90,2] + -21.524;
   1:  PR[91,3] = PR[90,3] + 78.829;
   1:L PR[91] R[100]mm/sec CNT100;
   1:  PR[91,1] = PR[90,1] + 57.560;
   1:  PR[91,2] = PR[90,2] + -20.498;
   1:  PR[91,3] = PR[90,3] + 78.837;
   1:L PR[91] R[100]mm/sec CNT100;
   1:  PR[91,1] = PR[90,1] + 59.786;
   1:  PR[91,2] = PR[90,2] + -19.072;
   1:  PR[91,3] = PR[90,3] + 78.843;
   1:L PR[91] R[100]mm/sec CNT100;
   1:  PR[91,1] = PR[90,1] + 62.571;
   1:  PR[91,2] = PR[90,2] + -16.719;
   1:  PR[91,3] = PR[90,3] + 78.854;
   1:L PR[91] R[100]mm/sec CNT100;
   1:  PR[91,1] = PR[90,1] + 63.263;
   1:  PR[91,2] = PR[90,2] + -16.116;
   1:  PR[91,3] = PR[90,3] + 78.868;
   1:L PR[91] R[100]mm/sec CNT100;
   1:  PR[91,1] = PR[90,1] + 63.827;
   1:  PR[91,2] = PR[90,2] + -15.457;
   1:  PR[91,3] = PR[90,3] + 78.872;
   1:L PR[91] R[100]mm/sec CNT100;
   1:  PR[91,1] = PR[90,1] + 66.315;
   1:  PR[91,2] = PR[90,2] + -12.369;
   1:  PR[91,3] = PR[90,3] + 78.875;
   1:L PR[91] R[100]mm/sec CNT100;
   1:  PR[91,1] = PR[90,1] + 67.947;
   1:  PR[91,2] = PR[90,2] + -9.434;
   1:  PR[91,3] = PR[90,3] + 78.890;
   1:L PR[91] R[100]mm/sec CNT100;
   1:  PR[91,1] = PR[90,1] + 68.606;
   1:  PR[91,2] = PR[90,2] + -7.928;
   1:  PR[91,3] = PR[90,3] + 78.904;
   1:L PR[91] R[100]mm/sec CNT100;
   1:  PR[91,1] = PR[90,1] + 69.456;
   1:  PR[91,2] = PR[90,2] + -5.289;
   1:  PR[91,3] = PR[90,3] + 78.910;
   1:L PR[91] R[100]mm/sec CNT100;
   1:  PR[91,1] = PR[90,1] + 69.757;
   1:  PR[91,2] = PR[90,2] + -3.183;
   1:  PR[91,3] = PR[90,3] + 78.921;
   1:L PR[91] R[100]mm/sec CNT100;
   1:  PR[91,1] = PR[90,1] + 70.012;
   1:  PR[91,2] = PR[90,2] + -0.768;
   1:  PR[91,3] = PR[90,3] + 78.929;
   1:L PR[91] R[100]mm/sec CNT100;
   1:  PR[91,1] = PR[90,1] + 69.706;
   1:  PR[91,2] = PR[90,2] + 1.349;
   1:  PR[91,3] = PR[90,3] + 78.939;
   1:L PR[91] R[100]mm/sec CNT100;
   1:  PR[91,1] = PR[90,1] + 69.445;
   1:  PR[91,2] = PR[90,2] + 3.866;
   1:  PR[91,3] = PR[90,3] + 78.947;
   1:L PR[91] R[100]mm/sec CNT100;
   1:  PR[91,1] = PR[90,1] + 68.606;
   1:  PR[91,2] = PR[90,2] + 6.468;
   1:  PR[91,3] = PR[90,3] + 78.957;
   1:L PR[91] R[100]mm/sec CNT100;
   1:  PR[91,1] = PR[90,1] + 67.947;
